	X =  251.204  mm,	Y =   -385.900  mm,	Z =   -311.265  mm,
	W =  90.000 deg,	P =   0.000 deg,	R =   90.000 deg
};
P[2440]{
   GP1:
	UF : 0, UT : 6,		CONFIG : 'N U T, 0, 0, 0',
	X =  250.053  mm,	Y =   -385.942  mm,	Z =   -320.068  mm,
	W =  90.000 deg,	P =   0.000 deg,	R =   90.000 deg
};
P[2441]{
   GP1:
	UF : 0, UT : 6,		CONFIG : 'N U T, 0, 0, 0',
	X =  249.566  mm,	Y =   -387.016  mm,	Z =   -309.000  mm,
	W =  90.000 deg,	P =   0.000 deg,	R =   90.000 deg
};
P[2442]{
   GP1:
	UF : 0, UT : 6,		CONFIG : 'N U T, 0, 0, 0',
	X =  248.771  mm,	Y =   -387.237  mm,	Z =   -309.100  mm,
	W =  90.000 deg,	P =   0.000 deg,	R =   90.000 deg
};
P[2443]{
   GP1:
	UF : 0, UT : 6,		CONFIG : 'N U T, 0, 0, 0',
	X =  247.127  mm,	Y =   -387.817  mm,	Z =   -310.009  mm,
	W =  90.000 deg,	P =   0.000 deg,	R =   90.000 deg
};
P[2444]{
   GP1:
	UF : 0, UT : 6,		CONFIG : 'N U T, 0, 0, 0',
	X =  246.328  mm,	Y =   -388.859  mm,	Z =   -309.000  mm,
	W =  90.000 deg,	P =   0.000 deg,	R =   90.000 deg
};
P[2445]{
   GP1:
	UF : 0, UT : 6,		CONFIG : 'N U T, 0, 0, 0',
	X =  245.729  mm,	Y =   -389.069  mm,	Z =   -324.841  mm,
	W =  90.000 deg,	P =   0.000 deg,	R =   90.000 deg
};
P[2446]{
   GP1:
	UF : 0, UT : 6,		CONFIG : 'N U T, 0, 0, 0',
	X =  244.982  mm,	Y =   -389.746  mm,	Z =   -309.100  mm,
	W =  90.000 deg,	P =   0.000 deg,	R =   90.000 deg
};
P[2447]{
   GP1:
	UF : 0, UT : 6,		CONFIG : 'N U T, 0, 0, 0',
	X =  243.856  mm,	Y =   -389.819  mm,	Z =   -309.100  mm,
	W =  90.000 deg,	P =   0.000 deg,	R =   90.000 deg
};
P[2448]{
   GP1:
	UF : 0, UT : 6,		CONFIG : 'N U T, 0, 0, 0',
	X =  243.235  mm,	Y =   -390.864  mm,	Z =   -309.100  mm,
	W =  90.000 deg,	P =   0.000 deg,	R =   90.000 deg
};
P[2449]{
   GP1:
	UF : 0, UT : 6,		CONFIG : 'N U T, 0, 0, 0',
	X =  242.193  mm,	Y =   -390.693  mm,	Z =   -309.000  mm,
	W =  90.000 deg,	P =   0.000 deg,	R =   90.000 deg
};
P[2450]{
   GP1:
	UF : 0, UT : 6,		CONFIG : 'N U T, 0, 0, 0',
	X =  241.203  mm,	Y =   -391.822  mm,	Z =   -309.100  mm,
	W =  90.000 deg,	P =   0.000 deg,	R =   90.000 deg
};
P[2451]{
   GP1:
	UF : 0, UT : 6,		CONFIG : 'N U T, 0, 0, 0',
	X =  240.398  mm,	Y =   -392.107  mm,	Z =   -309.000  mm,
	W =  90.000 deg,	P =   0.000 deg,	R =   90.000 deg
};
P[2452]{
   GP1:
	UF : 0, UT : 6,		CONFIG : 'N U T, 0, 0, 0',
	X =  239.660  mm,	Y =   -391.959  mm,	Z =   -309.100  mm,
	W =  90.000 deg,	P =   0.000 deg,	R =   90.000 deg
};
P[2453]{
   GP1:
	UF : 0, UT : 6,		CONFIG : 'N U T, 0, 0, 0',
	X =  238.993  mm,	Y =   -392.564  mm,	Z =   -309.000  mm,
	W =  90.000 deg,	P =   0.000 deg,	R =   90.000 deg
};
P[2454]{
   GP1:
	UF : 0, UT : 6,		CONFIG : 'N U T, 0, 0, 0',
	X =  238.146  mm,	Y =   -393.472  mm,	Z =   -309.000  mm,
	W =  90.000 deg,	P =   0.000 deg,	R =   90.000 deg
};
P[2455]{
   GP1:
	UF : 0, UT : 6,		CONFIG : 'N U T, 0, 0, 0',
	X =  236.954  mm,	Y =   -394.057  mm,	Z =   -309.000  mm,
	W =  90.000 deg,	P =   0.000 deg,	R =   90.000 deg
};
P[2456]{
   GP1:
	UF : 0, UT : 6,		CONFIG : 'N U T, 0, 0, 0',
	X =  236.048  mm,	Y =   -394.584  mm,	Z =   -309.100  mm,
	W =  90.000 deg,	P =   0.000 deg,	R =   90.000 deg
};
P[2457]{
   GP1:
	UF : 0, UT : 6,		CONFIG : 'N U T, 0, 0, 0',
	X =  235.652  mm,	Y =   -394.509  mm,	Z =   -309.100  mm,
	W =  90.000 deg,	P =   0.000 deg,	R =   90.000 deg
};
P[2458]{
   GP1:
	UF : 0, UT : 6,		CONFIG : 'N U T, 0, 0, 0',
	X =  235.672  mm,	Y =   -394.578  mm,	Z =   -309.000  mm,
	W =  90.000 deg,	P =   0.000 deg,	R =   90.000 deg
};
P[2459]{
   GP1:
	UF : 0, UT : 6,		CONFIG : 'N U T, 0, 0, 0',
	X =  235.717  mm,	Y =   -394.656  mm,	Z =   -309.100  mm,
	W =  90.000 deg,	P =   0.000 deg,	R =   90.000 deg
};
P[2460]{
   GP1:
	UF : 0, UT : 6,		CONFIG : 'N U T, 0, 0, 0',
	X =  235.797  mm,	Y =   -394.793  mm,	Z =   -309.100  mm,
	W =  90.000 deg,	P =   0.000 deg,	R =   90.000 deg
};
P[2461]{
   GP1:
	UF : 0, UT : 6,		CONFIG : 'N U T, 0, 0, 0',
	X =  235.811  mm,	Y =   -394.818  mm,	Z =   -309.000  mm,
	W =  90.000 deg,	P =   0.000 deg,	R =   90.000 deg
};
P[2462]{
   GP1:
	UF : 0, UT : 6,		CONFIG : 'N U T, 0, 0, 0',
	X =  235.830  mm,	Y =   -394.850  mm,	Z =   -309.000  mm,
	W =  90.000 deg,	P =   0.000 deg,	R =   90.000 deg
};
P[2463]{
   GP1:
	UF : 0, UT : 6,		CONFIG : 'N U T, 0, 0, 0',
	X =  235.853  mm,	Y =   -394.890  mm,	Z =   -309.000  mm,
	W =  90.000 deg,	P =   0.000 deg,	R =   90.000 deg
};
P[2464]{
   GP1:
	UF : 0, UT : 6,		CONFIG : 'N U T, 0, 0, 0',
	X =  235.853  mm,	Y =   -394.890  mm,	Z =   -309.100  mm,
	W =  90.000 deg,	P =   0.000 deg,	R =   90.000 deg
};
P[2465]{
   GP1:
	UF : 0, UT : 6,		CONFIG : 'N U T, 0, 0, 0',
	X =  235.932  mm,	Y =   -395.027  mm,	Z =   -309.000  mm,
	W =  90.000 deg,	P =   0.000 deg,	R =   90.000 deg
};
P[2466]{
   GP1:
	UF : 0, UT : 6,		CONFIG : 'N U T, 0, 0, 0',
	X =  234.712  mm,	Y =   -395.169  mm,	Z =   -311.663  mm,
	W =  90.000 deg,	P =   0.000 deg,	R =   90.000 deg
};
P[2467]{
   GP1:
	UF : 0, UT : 6,		CONFIG : 'N U T, 0, 0, 0',
	X =  233.900  mm,	Y =   -396.049  mm,	Z =   -309.000  mm,
	W =  90.000 deg,	P =   0.000 deg,	R =   90.000 deg
};
P[2468]{
   GP1:
	UF : 0, UT : 6,		CONFIG : 'N U T, 0, 0, 0',
	X =  232.847  mm,	Y =   -396.367  mm,	Z =   -309.000  mm,
	W =  90.000 deg,	P =   0.000 deg,	R =   90.000 deg
};
P[2469]{
   GP1:
	UF : 0, UT : 6,		CONFIG : 'N U T, 0, 0, 0',
	X =  231.860  mm,	Y =   -397.593  mm,	Z =   -322.086  mm,
	W =  90.000 deg,	P =   0.000 deg,	R =   90.000 deg
};
P[2470]{
   GP1:
	UF : 0, UT : 6,		CONFIG : 'N U T, 0, 0, 0',
	X =  231.255  mm,	Y =   -396.883  mm,	Z =   -309.100  mm,
	W =  90.000 deg,	P =   0.000 deg,	R =   90.000 deg
};
P[2471]{
   GP1:
	UF : 0, UT : 6,		CONFIG : 'N U T, 0, 0, 0',
	X =  230.508  mm,	Y =   -398.026  mm,	Z =   -309.100  mm,
	W =  90.000 deg,	P =   0.000 deg,	R =   90.000 deg
};
P[2472]{
   GP1:
	UF : 0, UT : 6,		CONFIG : 'N U T, 0, 0, 0',
	X =  229.295  mm,	Y =   -398.480  mm,	Z =   -309.000  mm,
	W =  90.000 deg,	P =   0.000 deg,	R =   90.000 deg
};
P[2473]{
   GP1:
	UF : 0, UT : 6,		CONFIG : 'N U T, 0, 0, 0',
	X =  228.271  mm,	Y =   -399.037  mm,	Z =   -309.100  mm,
	W =  90.000 deg,	P =   0.000 deg,	R =   90.000 deg
};
P[2474]{
   GP1:
	UF : 0, UT : 6,		CONFIG : 'N U T, 0, 0, 0',
	X =  227.431  mm,	Y =   -399.645  mm,	Z =   -309.000  mm,
	W =  90.000 deg,	P =   0.000 deg,	R =   90.000 deg
};
P[2475]{
   GP1:
	UF : 0, UT : 6,		CONFIG : 'N U T, 0, 0, 0',
	X =  227.107  mm,	Y =   -400.328  mm,	Z =   -309.000  mm,
	W =  90.000 deg,	P =   0.000 deg,	R =   90.000 deg
};
P[2476]{
   GP1:
	UF : 0, UT : 6,		CONFIG : 'N U T, 0, 0, 0',
	X =  226.158  mm,	Y =   -400.362  mm,	Z =   -309.000  mm,
	W =  90.000 deg,	P =   0.000 deg,	R =   90.000 deg
};
P[2477]{
   GP1:
	UF : 0, UT : 6,		CONFIG : 'N U T, 0, 0, 0',
	X =  225.458  mm,	Y =   -400.942  mm,	Z =   -309.100  mm,
	W =  90.000 deg,	P =   0.000 deg,	R =   90.000 deg
};
P[2478]{
   GP1:
	UF : 0, UT : 6,		CONFIG : 'N U T, 0, 0, 0',
	X =  223.961  mm,	Y =   -401.723  mm,	Z =   -309.000  mm,
	W =  90.000 deg,	P =   0.000 deg,	R =   90.000 deg
};
P[2479]{
   GP1:
	UF : 0, UT : 6,		CONFIG : 'N U T, 0, 0, 0',
	X =  222.266  mm,	Y =   -402.738  mm,	Z =   -309.000  mm,
	W =  90.000 deg,	P =   0.000 deg,	R =   90.000 deg
};
P[2480]{
   GP1:
	UF : 0, UT : 6,		CONFIG : 'N U T, 0, 0, 0',
	X =  221.544  mm,	Y =   -403.115  mm,	Z =   -309.000  mm,
	W =  90.000 deg,	P =   0.000 deg,	R =   90.000 deg
};
P[2481]{
   GP1:
	UF : 0, UT : 6,		CONFIG : 'N U T, 0, 0, 0',
	X =  220.694  mm,	Y =   -403.242  mm,	Z =   -309.100  mm,
	W =  90.000 deg,	P =   0.000 deg,	R =   90.000 deg
};
P[2482]{
   GP1:
	UF : 0, UT : 6,		CONFIG : 'N U T, 0, 0, 0',
	X =  220.123  mm,	Y =   -403.736  mm,	Z =   -309.000  mm,
	W =  90.000 deg,	P =   0.000 deg,	R =   90.000 deg
};
P[2483]{
   GP1:
	UF : 0, UT : 6,		CONFIG : 'N U T, 0, 0, 0',
	X =  218.860  mm,	Y =   -404.272  mm,	Z =   -309.000  mm,
	W =  90.000 deg,	P =   0.000 deg,	R =   90.000 deg
};
P[2484]{
   GP1:
	UF : 0, UT : 6,		CONFIG : 'N U T, 0, 0, 0',
	X =  217.826  mm,	Y =   -405.083  mm,	Z =   -309.000  mm,
	W =  90.000 deg,	P =   0.000 deg,	R =   90.000 deg
};
P[2485]{
   GP1:
	UF : 0, UT : 6,		CONFIG : 'N U T, 0, 0, 0',
	X =  217.425  mm,	Y =   -405.654  mm,	Z =   -309.100  mm,
	W =  90.000 deg,	P =   0.000 deg,	R =   90.000 deg
};
P[2486]{
   GP1:
	UF : 0, UT : 6,		CONFIG : 'N U T, 0, 0, 0',
	X =  216.186  mm,	Y =   -405.730  mm,	Z =   -309.000  mm,
	W =  90.000 deg,	P =   0.000 deg,	R =   90.000 deg
};
P[2487]{
   GP1:
	UF : 0, UT : 6,		CONFIG : 'N U T, 0, 0, 0',
	X =  215.322  mm,	Y =   -406.588  mm,	Z =   -309.000  mm,
	W =  90.000 deg,	P =   0.000 deg,	R =   90.000 deg
};
P[2488]{
   GP1:
	UF : 0, UT : 6,		CONFIG : 'N U T, 0, 0, 0',
	X =  214.425  mm,	Y =   -406.938  mm,	Z =   -309.000  mm,
	W =  90.000 deg,	P =   0.000 deg,	R =   90.000 deg
};
P[2489]{
   GP1:
	UF : 0, UT : 6,		CONFIG : 'N U T, 0, 0, 0',
	X =  212.907  mm,	Y =   -407.890  mm,	Z =   -309.000  mm,
	W =  90.000 deg,	P =   0.000 deg,	R =   90.000 deg
};
P[2490]{
   GP1:
	UF : 0, UT : 6,		CONFIG : 'N U T, 0, 0, 0',
	X =  212.273  mm,	Y =   -408.822  mm,	Z =   -309.000  mm,
	W =  90.000 deg,	P =   0.000 deg,	R =   90.000 deg
};
P[2491]{
   GP1:
	UF : 0, UT : 6,		CONFIG : 'N U T, 0, 0, 0',
	X =  211.523  mm,	Y =   -408.247  mm,	Z =   -309.840  mm,
	W =  90.000 deg,	P =   0.000 deg,	R =   90.000 deg
};
P[2492]{
   GP1:
	UF : 0, UT : 6,		CONFIG : 'N U T, 0, 0, 0',
	X =  211.810  mm,	Y =   -408.899  mm,	Z =   -309.000  mm,
	W =  90.000 deg,	P =   0.000 deg,	R =   90.000 deg
};
P[2493]{
   GP1:
	UF : 0, UT : 6,		CONFIG : 'N U T, 0, 0, 0',
	X =  211.264  mm,	Y =   -408.563  mm,	Z =   -309.000  mm,
	W =  90.000 deg,	P =   0.000 deg,	R =   90.000 deg
};
P[2494]{
   GP1:
	UF : 0, UT : 6,		CONFIG : 'N U T, 0, 0, 0',
	X =  211.213  mm,	Y =   -409.187  mm,	Z =   -309.100  mm,
	W =  90.000 deg,	P =   0.000 deg,	R =   90.000 deg
};
P[2495]{
   GP1:
	UF : 0, UT : 6,		CONFIG : 'N U T, 0, 0, 0',
	X =  210.542  mm,	Y =   -409.005  mm,	Z =   -309.000  mm,
	W =  90.000 deg,	P =   0.000 deg,	R =   90.000 deg
};
P[2496]{
   GP1:
	UF : 0, UT : 6,		CONFIG : 'N U T, 0, 0, 0',
	X =  210.183  mm,	Y =   -409.615  mm,	Z =   -311.087  mm,
	W =  90.000 deg,	P =   0.000 deg,	R =   90.000 deg
};
P[2497]{
   GP1:
	UF : 0, UT : 6,		CONFIG : 'N U T, 0, 0, 0',
	X =  209.312  mm,	Y =   -409.801  mm,	Z =   -309.000  mm,
	W =  90.000 deg,	P =   0.000 deg,	R =   90.000 deg
};
P[2498]{
   GP1:
	UF : 0, UT : 6,		CONFIG : 'N U T, 0, 0, 0',
	X =  208.830  mm,	Y =   -410.582  mm,	Z =   -326.834  mm,
	W =  90.000 deg,	P =   0.000 deg,	R =   90.000 deg
};
P[2499]{
   GP1:
	UF : 0, UT : 6,		CONFIG : 'N U T, 0, 0, 0',
	X =  207.578  mm,	Y =   -411.271  mm,	Z =   -319.896  mm,
	W =  90.000 deg,	P =   0.000 deg,	R =   90.000 deg
};
P[2500]{
   GP1:
	UF : 0, UT : 6,		CONFIG : 'N U T, 0, 0, 0',
	X =  206.272  mm,	Y =   -411.225  mm,	Z =   -309.000  mm,
	W =  90.000 deg,	P =   0.000 deg,	R =   90.000 deg
};
P[2501]{
   GP1:
	UF : 0, UT : 6,		CONFIG : 'N U T, 0, 0, 0',
	X =  205.768  mm,	Y =   -411.902  mm,	Z =   -309.000  mm,
	W =  90.000 deg,	P =   0.000 deg,	R =   90.000 deg
};
P[2502]{
   GP1:
	UF : 0, UT : 6,		CONFIG : 'N U T, 0, 0, 0',
	X =  205.135  mm,	Y =   -412.565  mm,	Z =   -309.000  mm,
	W =  90.000 deg,	P =   0.000 deg,	R =   90.000 deg
};
P[2503]{
   GP1:
	UF : 0, UT : 6,		CONFIG : 'N U T, 0, 0, 0',
	X =  204.079  mm,	Y =   -412.679  mm,	Z =   -309.000  mm,
	W =  90.000 deg,	P =   0.000 deg,	R =   90.000 deg
};
P[2504]{
   GP1:
	UF : 0, UT : 6,		CONFIG : 'N U T, 0, 0, 0',
	X =  203.955  mm,	Y =   -413.351  mm,	Z =   -309.000  mm,
	W =  90.000 deg,	P =   0.000 deg,	R =   90.000 deg
};
P[2505]{
   GP1:
	UF : 0, UT : 6,		CONFIG : 'N U T, 0, 0, 0',
	X =  203.212  mm,	Y =   -413.679  mm,	Z =   -309.100  mm,
	W =  90.000 deg,	P =   0.000 deg,	R =   90.000 deg
};
P[2506]{
   GP1:
	UF : 0, UT : 6,		CONFIG : 'N U T, 0, 0, 0',
	X =  201.743  mm,	Y =   -414.498  mm,	Z =   -320.312  mm,
	W =  90.000 deg,	P =   0.000 deg,	R =   90.000 deg
};
P[2507]{
   GP1:
	UF : 0, UT : 6,		CONFIG : 'N U T, 0, 0, 0',
	X =  200.955  mm,	Y =   -414.995  mm,	Z =   -309.100  mm,
	W =  90.000 deg,	P =   0.000 deg,	R =   90.000 deg
};
P[2508]{
   GP1:
	UF : 0, UT : 6,		CONFIG : 'N U T, 0, 0, 0',
	X =  199.958  mm,	Y =   -415.276  mm,	Z =   -309.000  mm,
	W =  90.000 deg,	P =   0.000 deg,	R =   90.000 deg
};
P[2509]{
   GP1:
	UF : 0, UT : 6,		CONFIG : 'N U T, 0, 0, 0',
	X =  199.292  mm,	Y =   -415.680  mm,	Z =   -309.000  mm,
	W =  90.000 deg,	P =   0.000 deg,	R =   90.000 deg
};
P[2510]{
   GP1:
	UF : 0, UT : 6,		CONFIG : 'N U T, 0, 0, 0',
	X =  198.614  mm,	Y =   -416.039  mm,	Z =   -309.000  mm,
	W =  90.000 deg,	P =   0.000 deg,	R =   90.000 deg
};
P[2511]{
   GP1:
	UF : 0, UT : 6,		CONFIG : 'N U T, 0, 0, 0',
	X =  197.853  mm,	Y =   -416.086  mm,	Z =   -309.100  mm,
	W =  90.000 deg,	P =   0.000 deg,	R =   90.000 deg
};
P[2512]{
   GP1:
	UF : 0, UT : 6,		CONFIG : 'N U T, 0, 0, 0',
	X =  197.431  mm,	Y =   -416.630  mm,	Z =   -309.000  mm,
	W =  90.000 deg,	P =   0.000 deg,	R =   90.000 deg
};
P[2513]{
   GP1:
	UF : 0, UT : 6,		CONFIG : 'N U T, 0, 0, 0',
	X =  197.048  mm,	Y =   -417.376  mm,	Z =   -309.000  mm,
	W =  90.000 deg,	P =   0.000 deg,	R =   90.000 deg
};
P[2514]{
   GP1:
	UF : 0, UT : 6,		CONFIG : 'N U T, 0, 0, 0',
	X =  195.899  mm,	Y =   -417.317  mm,	Z =   -309.100  mm,
	W =  90.000 deg,	P =   0.000 deg,	R =   90.000 deg
};
P[2515]{
   GP1:
	UF : 0, UT : 6,		CONFIG : 'N U T, 0, 0, 0',
	X =  195.162  mm,	Y =   -418.086  mm,	Z =   -309.769  mm,
	W =  90.000 deg,	P =   0.000 deg,	R =   90.000 deg
};
P[2516]{
   GP1:
	UF : 0, UT : 6,		CONFIG : 'N U T, 0, 0, 0',
	X =  193.868  mm,	Y =   -419.148  mm,	Z =   -320.299  mm,
	W =  90.000 deg,	P =   0.000 deg,	R =   90.000 deg
};
P[2517]{
   GP1:
	UF : 0, UT : 6,		CONFIG : 'N U T, 0, 0, 0',
	X =  192.981  mm,	Y =   -419.724  mm,	Z =   -309.000  mm,
	W =  90.000 deg,	P =   0.000 deg,	R =   90.000 deg
};
P[2518]{
   GP1:
	UF : 0, UT : 6,		CONFIG : 'N U T, 0, 0, 0',
	X =  191.775  mm,	Y =   -420.224  mm,	Z =   -309.100  mm,
	W =  90.000 deg,	P =   0.000 deg,	R =   90.000 deg
};
P[2519]{
   GP1:
	UF : 0, UT : 6,		CONFIG : 'N U T, 0, 0, 0',
	X =  190.726  mm,	Y =   -420.304  mm,	Z =   -309.000  mm,
	W =  90.000 deg,	P =   0.000 deg,	R =   90.000 deg
};
P[2520]{
   GP1:
	UF : 0, UT : 6,		CONFIG : 'N U T, 0, 0, 0',
	X =  191.173  mm,	Y =   -421.086  mm,	Z =   -309.000  mm,
	W =  90.000 deg,	P =   0.000 deg,	R =   90.000 deg
};
P[2521]{
   GP1:
	UF : 0, UT : 6,		CONFIG : 'N U T, 0, 0, 0',
	X =  190.334  mm,	Y =   -421.290  mm,	Z =   -322.014  mm,
	W =  90.000 deg,	P =   0.000 deg,	R =   90.000 deg
};
P[2522]{
   GP1:
	UF : 0, UT : 6,		CONFIG : 'N U T, 0, 0, 0',
	X =  189.270  mm,	Y =   -421.536  mm,	Z =   -309.000  mm,
	W =  90.000 deg,	P =   0.000 deg,	R =   90.000 deg
};
P[2523]{
   GP1:
	UF : 0, UT : 6,		CONFIG : 'N U T, 0, 0, 0',
	X =  187.988  mm,	Y =   -422.472  mm,	Z =   -309.000  mm,
	W =  90.000 deg,	P =   0.000 deg,	R =   90.000 deg
};
P[2524]{
   GP1:
	UF : 0, UT : 6,		CONFIG : 'N U T, 0, 0, 0',
	X =  186.884  mm,	Y =   -422.846  mm,	Z =   -309.000  mm,
	W =  90.000 deg,	P =   0.000 deg,	R =   90.000 deg
};
P[2525]{
   GP1:
	UF : 0, UT : 6,		CONFIG : 'N U T, 0, 0, 0',
	X =  186.127  mm,	Y =   -423.764  mm,	Z =   -309.000  mm,
	W =  90.000 deg,	P =   0.000 deg,	R =   90.000 deg
};
P[2526]{
   GP1:
	UF : 0, UT : 6,		CONFIG : 'N U T, 0, 0, 0',
	X =  184.971  mm,	Y =   -424.213  mm,	Z =   -309.000  mm,
	W =  90.000 deg,	P =   0.000 deg,	R =   90.000 deg
};
P[2527]{
   GP1:
	UF : 0, UT : 6,		CONFIG : 'N U T, 0, 0, 0',
	X =  184.314  mm,	Y =   -424.591  mm,	Z =   -309.000  mm,
	W =  90.000 deg,	P =   0.000 deg,	R =   90.000 deg
};
P[2528]{
   GP1:
	UF : 0, UT : 6,		CONFIG : 'N U T, 0, 0, 0',
	X =  182.781  mm,	Y =   -425.363  mm,	Z =   -309.000  mm,
	W =  90.000 deg,	P =   0.000 deg,	R =   90.000 deg
};
P[2529]{
   GP1:
	UF : 0, UT : 6,		CONFIG : 'N U T, 0, 0, 0',
	X =  181.660  mm,	Y =   -425.576  mm,	Z =   -309.100  mm,
	W =  90.000 deg,	P =   0.000 deg,	R =   90.000 deg
};
P[2530]{
   GP1:
	UF : 0, UT : 6,		CONFIG : 'N U T, 0, 0, 0',
	X =  181.249  mm,	Y =   -426.623  mm,	Z =   -309.000  mm,
	W =  90.000 deg,	P =   0.000 deg,	R =   90.000 deg
};
P[2531]{
   GP1:
	UF : 0, UT : 6,		CONFIG : 'N U T, 0, 0, 0',
	X =  180.447  mm,	Y =   -426.800  mm,	Z =   -309.000  mm,
	W =  90.000 deg,	P =   0.000 deg,	R =   90.000 deg
};
P[2532]{
   GP1:
	UF : 0, UT : 6,		CONFIG : 'N U T, 0, 0, 0',
	X =  179.771  mm,	Y =   -426.566  mm,	Z =   -309.000  mm,
	W =  90.000 deg,	P =   0.000 deg,	R =   90.000 deg
};
P[2533]{
   GP1:
	UF : 0, UT : 6,		CONFIG : 'N U T, 0, 0, 0',
	X =  179.286  mm,	Y =   -427.366  mm,	Z =   -309.000  mm,
	W =  90.000 deg,	P =   0.000 deg,	R =   90.000 deg
};
P[2534]{
   GP1:
	UF : 0, UT : 6,		CONFIG : 'N U T, 0, 0, 0',
	X =  178.106  mm,	Y =   -427.866  mm,	Z =   -309.100  mm,
	W =  90.000 deg,	P =   0.000 deg,	R =   90.000 deg
};
P[2535]{
   GP1:
	UF : 0, UT : 6,		CONFIG : 'N U T, 0, 0, 0',
	X =  177.596  mm,	Y =   -428.277  mm,	Z =   -309.000  mm,
	W =  90.000 deg,	P =   0.000 deg,	R =   90.000 deg
};
P[2536]{
   GP1:
	UF : 0, UT : 6,		CONFIG : 'N U T, 0, 0, 0',
	X =  176.414  mm,	Y =   -428.917  mm,	Z =   -309.000  mm,
	W =  90.000 deg,	P =   0.000 deg,	R =   90.000 deg
};
P[2537]{
   GP1:
	UF : 0, UT : 6,		CONFIG : 'N U T, 0, 0, 0',
	X =  175.410  mm,	Y =   -429.586  mm,	Z =   -309.000  mm,
	W =  90.000 deg,	P =   0.000 deg,	R =   90.000 deg
};
P[2538]{
   GP1:
	UF : 0, UT : 6,		CONFIG : 'N U T, 0, 0, 0',
	X =  174.790  mm,	Y =   -430.203  mm,	Z =   -309.100  mm,
	W =  90.000 deg,	P =   0.000 deg,	R =   90.000 deg
};
P[2539]{
   GP1:
	UF : 0, UT : 6,		CONFIG : 'N U T, 0, 0, 0',
	X =  174.023  mm,	Y =   -430.329  mm,	Z =   -309.000  mm,
	W =  90.000 deg,	P =   0.000 deg,	R =   90.000 deg
};
P[2540]{
   GP1:
	UF : 0, UT : 6,		CONFIG : 'N U T, 0, 0, 0',
	X =  173.246  mm,	Y =   -430.866  mm,	Z =   -309.000  mm,
	W =  90.000 deg,	P =   0.000 deg,	R =   90.000 deg
};
P[2541]{
   GP1:
	UF : 0, UT : 6,		CONFIG : 'N U T, 0, 0, 0',
	X =  172.207  mm,	Y =   -431.345  mm,	Z =   -309.000  mm,
	W =  90.000 deg,	P =   0.000 deg,	R =   90.000 deg
};
P[2542]{
   GP1:
	UF : 0, UT : 6,		CONFIG : 'N U T, 0, 0, 0',
	X =  171.867  mm,	Y =   -432.022  mm,	Z =   -309.000  mm,
	W =  90.000 deg,	P =   0.000 deg,	R =   90.000 deg
};
P[2543]{
   GP1:
	UF : 0, UT : 6,		CONFIG : 'N U T, 0, 0, 0',
	X =  170.157  mm,	Y =   -432.977  mm,	Z =   -309.000  mm,
	W =  90.000 deg,	P =   0.000 deg,	R =   90.000 deg
};
P[2544]{
   GP1:
	UF : 0, UT : 6,		CONFIG : 'N U T, 0, 0, 0',
	X =  169.135  mm,	Y =   -432.828  mm,	Z =   -309.000  mm,
	W =  90.000 deg,	P =   0.000 deg,	R =   90.000 deg
};
P[2545]{
   GP1:
	UF : 0, UT : 6,		CONFIG : 'N U T, 0, 0, 0',
	X =  168.495  mm,	Y =   -433.303  mm,	Z =   -309.000  mm,
	W =  90.000 deg,	P =   0.000 deg,	R =   90.000 deg
};
P[2546]{
   GP1:
	UF : 0, UT : 6,		CONFIG : 'N U T, 0, 0, 0',
	X =  168.424  mm,	Y =   -434.070  mm,	Z =   -309.000  mm,
	W =  90.000 deg,	P =   0.000 deg,	R =   90.000 deg
};
P[2547]{
   GP1:
	UF : 0, UT : 6,		CONFIG : 'N U T, 0, 0, 0',
	X =  166.498  mm,	Y =   -434.623  mm,	Z =   -309.000  mm,
	W =  90.000 deg,	P =   0.000 deg,	R =   90.000 deg
};
P[2548]{
   GP1:
	UF : 0, UT : 6,		CONFIG : 'N U T, 0, 0, 0',
	X =  165.399  mm,	Y =   -435.440  mm,	Z =   -309.000  mm,
	W =  90.000 deg,	P =   0.000 deg,	R =   90.000 deg
};
P[2549]{
   GP1:
	UF : 0, UT : 6,		CONFIG : 'N U T, 0, 0, 0',
	X =  164.602  mm,	Y =   -435.687  mm,	Z =   -309.000  mm,
	W =  90.000 deg,	P =   0.000 deg,	R =   90.000 deg
};
P[2550]{
   GP1:
	UF : 0, UT : 6,		CONFIG : 'N U T, 0, 0, 0',
	X =  163.906  mm,	Y =   -436.668  mm,	Z =   -309.000  mm,
	W =  90.000 deg,	P =   0.000 deg,	R =   90.000 deg
};
P[2551]{
   GP1:
	UF : 0, UT : 6,		CONFIG : 'N U T, 0, 0, 0',
	X =  162.841  mm,	Y =   -437.088  mm,	Z =   -309.100  mm,
	W =  90.000 deg,	P =   0.000 deg,	R =   90.000 deg
};
P[2552]{
   GP1:
	UF : 0, UT : 6,		CONFIG : 'N U T, 0, 0, 0',
	X =  161.989  mm,	Y =   -437.881  mm,	Z =   -309.893  mm,
	W =  90.000 deg,	P =   0.000 deg,	R =   90.000 deg
};
P[2553]{
   GP1:
	UF : 0, UT : 6,		CONFIG : 'N U T, 0, 0, 0',
	X =  161.304  mm,	Y =   -437.408  mm,	Z =   -309.000  mm,
	W =  90.000 deg,	P =   0.000 deg,	R =   90.000 deg
};
P[2554]{
   GP1:
	UF : 0, UT : 6,		CONFIG : 'N U T, 0, 0, 0',
	X =  160.368  mm,	Y =   -438.644  mm,	Z =   -309.000  mm,
	W =  90.000 deg,	P =   0.000 deg,	R =   90.000 deg
};
P[2555]{
   GP1:
	UF : 0, UT : 6,		CONFIG : 'N U T, 0, 0, 0',
	X =  159.528  mm,	Y =   -438.648  mm,	Z =   -309.000  mm,
	W =  90.000 deg,	P =   0.000 deg,	R =   90.000 deg
};
P[2556]{
   GP1:
	UF : 0, UT : 6,		CONFIG : 'N U T, 0, 0, 0',
	X =  158.573  mm,	Y =   -439.371  mm,	Z =   -309.000  mm,
	W =  90.000 deg,	P =   0.000 deg,	R =   90.000 deg
};
P[2557]{
   GP1:
	UF : 0, UT : 6,		CONFIG : 'N U T, 0, 0, 0',
	X =  157.879  mm,	Y =   -440.242  mm,	Z =   -309.000  mm,
	W =  90.000 deg,	P =   0.000 deg,	R =   90.000 deg
};
P[2558]{
   GP1:
	UF : 0, UT : 6,		CONFIG : 'N U T, 0, 0, 0',
	X =  157.140  mm,	Y =   -440.386  mm,	Z =   -309.000  mm,
	W =  90.000 deg,	P =   0.000 deg,	R =   90.000 deg
};
P[2559]{
   GP1:
	UF : 0, UT : 6,		CONFIG : 'N U T, 0, 0, 0',
	X =  156.396  mm,	Y =   -440.305  mm,	Z =   -309.000  mm,
	W =  90.000 deg,	P =   0.000 deg,	R =   90.000 deg
};
P[2560]{
   GP1:
	UF : 0, UT : 6,		CONFIG : 'N U T, 0, 0, 0',
	X =  155.713  mm,	Y =   -441.118  mm,	Z =   -309.000  mm,
	W =  90.000 deg,	P =   0.000 deg,	R =   90.000 deg
};
P[2561]{
   GP1:
	UF : 0, UT : 6,		CONFIG : 'N U T, 0, 0, 0',
	X =  155.008  mm,	Y =   -441.324  mm,	Z =   -309.000  mm,
	W =  90.000 deg,	P =   0.000 deg,	R =   90.000 deg
};
P[2562]{
   GP1:
	UF : 0, UT : 6,		CONFIG : 'N U T, 0, 0, 0',
	X =  154.353  mm,	Y =   -441.739  mm,	Z =   -309.000  mm,
	W =  90.000 deg,	P =   0.000 deg,	R =   90.000 deg
};
P[2563]{
   GP1:
	UF : 0, UT : 6,		CONFIG : 'N U T, 0, 0, 0',
	X =  153.918  mm,	Y =   -442.344  mm,	Z =   -309.000  mm,
	W =  90.000 deg,	P =   0.000 deg,	R =   90.000 deg
};
P[2564]{
   GP1:
	UF : 0, UT : 6,		CONFIG : 'N U T, 0, 0, 0',
	X =  153.557  mm,	Y =   -442.273  mm,	Z =   -309.000  mm,
	W =  90.000 deg,	P =   0.000 deg,	R =   90.000 deg
};
P[2565]{
   GP1:
	UF : 0, UT : 6,		CONFIG : 'N U T, 0, 0, 0',
	X =  153.337  mm,	Y =   -441.968  mm,	Z =   -309.000  mm,
	W =  90.000 deg,	P =   0.000 deg,	R =   90.000 deg
};
P[2566]{
   GP1:
	UF : 0, UT : 6,		CONFIG : 'N U T, 0, 0, 0',
	X =  153.390  mm,	Y =   -442.061  mm,	Z =   -309.100  mm,
	W =  90.000 deg,	P =   0.000 deg,	R =   90.000 deg
};
P[2567]{
   GP1:
	UF : 0, UT : 6,		CONFIG : 'N U T, 0, 0, 0',
	X =  153.417  mm,	Y =   -442.107  mm,	Z =   -309.100  mm,
	W =  90.000 deg,	P =   0.000 deg,	R =   90.000 deg
};
P[2568]{
   GP1:
	UF : 0, UT : 6,		CONFIG : 'N U T, 0, 0, 0',
	X =  153.429  mm,	Y =   -442.129  mm,	Z =   -309.000  mm,
	W =  90.000 deg,	P =   0.000 deg,	R =   90.000 deg
};
P[2569]{
   GP1:
	UF : 0, UT : 6,		CONFIG : 'N U T, 0, 0, 0',
	X =  153.499  mm,	Y =   -442.250  mm,	Z =   -309.000  mm,
	W =  90.000 deg,	P =   0.000 deg,	R =   90.000 deg
};
P[2570]{
   GP1:
	UF : 0, UT : 6,		CONFIG : 'N U T, 0, 0, 0',
	X =  153.512  mm,	Y =   -442.271  mm,	Z =   -309.000  mm,
	W =  90.000 deg,	P =   0.000 deg,	R =   90.000 deg
};
P[2571]{
   GP1:
	UF : 0, UT : 6,		CONFIG : 'N U T, 0, 0, 0',
	X =  153.675  mm,	Y =   -442.554  mm,	Z =   -309.000  mm,
	W =  90.000 deg,	P =   0.000 deg,	R =   90.000 deg
};
P[2572]{
   GP1:
	UF : 0, UT : 6,		CONFIG : 'N U T, 0, 0, 0',
	X =  153.676  mm,	Y =   -442.556  mm,	Z =   -309.100  mm,
	W =  90.000 deg,	P =   0.000 deg,	R =   90.000 deg
};
P[2573]{
   GP1:
	UF : 0, UT : 6,		CONFIG : 'N U T, 0, 0, 0',
	X =  153.700  mm,	Y =   -442.598  mm,	Z =   -309.000  mm,
	W =  90.000 deg,	P =   0.000 deg,	R =   90.000 deg
};
P[2574]{
   GP1:
	UF : 0, UT : 6,		CONFIG : 'N U T, 0, 0, 0',
	X =  153.197  mm,	Y =   -442.479  mm,	Z =   -309.100  mm,
	W =  90.000 deg,	P =   0.000 deg,	R =   90.000 deg
};
P[2575]{
   GP1:
	UF : 0, UT : 6,		CONFIG : 'N U T, 0, 0, 0',
	X =  151.809  mm,	Y =   -442.696  mm,	Z =   -309.000  mm,
	W =  90.000 deg,	P =   0.000 deg,	R =   90.000 deg
};
P[2576]{
   GP1:
	UF : 0, UT : 6,		CONFIG : 'N U T, 0, 0, 0',
	X =  151.136  mm,	Y =   -443.692  mm,	Z =   -319.431  mm,
	W =  90.000 deg,	P =   0.000 deg,	R =   90.000 deg
};
P[2577]{
   GP1:
	UF : 0, UT : 6,		CONFIG : 'N U T, 0, 0, 0',
	X =  150.368  mm,	Y =   -444.081  mm,	Z =   -309.000  mm,
	W =  90.000 deg,	P =   0.000 deg,	R =   90.000 deg
};
P[2578]{
   GP1:
	UF : 0, UT : 6,		CONFIG : 'N U T, 0, 0, 0',
	X =  149.653  mm,	Y =   -444.476  mm,	Z =   -309.000  mm,
	W =  90.000 deg,	P =   0.000 deg,	R =   90.000 deg
};
P[2579]{
   GP1:
	UF : 0, UT : 6,		CONFIG : 'N U T, 0, 0, 0',
	X =  148.623  mm,	Y =   -444.808  mm,	Z =   -309.000  mm,
	W =  90.000 deg,	P =   0.000 deg,	R =   90.000 deg
};
P[2580]{
   GP1:
	UF : 0, UT : 6,		CONFIG : 'N U T, 0, 0, 0',
	X =  147.296  mm,	Y =   -446.099  mm,	Z =   -309.000  mm,
	W =  90.000 deg,	P =   0.000 deg,	R =   90.000 deg
};
P[2581]{
   GP1:
	UF : 0, UT : 6,		CONFIG : 'N U T, 0, 0, 0',
	X =  146.188  mm,	Y =   -446.215  mm,	Z =   -309.000  mm,
	W =  90.000 deg,	P =   0.000 deg,	R =   90.000 deg
};
P[2582]{
   GP1:
	UF : 0, UT : 6,		CONFIG : 'N U T, 0, 0, 0',
	X =  145.216  mm,	Y =   -446.906  mm,	Z =   -309.100  mm,
	W =  90.000 deg,	P =   0.000 deg,	R =   90.000 deg
};
P[2583]{
   GP1:
	UF : 0, UT : 6,		CONFIG : 'N U T, 0, 0, 0',
	X =  144.453  mm,	Y =   -447.564  mm,	Z =   -309.000  mm,
	W =  90.000 deg,	P =   0.000 deg,	R =   90.000 deg
};
P[2584]{
   GP1:
	UF : 0, UT : 6,		CONFIG : 'N U T, 0, 0, 0',
	X =  143.642  mm,	Y =   -447.566  mm,	Z =   -309.100  mm,
	W =  90.000 deg,	P =   0.000 deg,	R =   90.000 deg
};
P[2585]{
   GP1:
	UF : 0, UT : 6,		CONFIG : 'N U T, 0, 0, 0',
	X =  142.855  mm,	Y =   -448.215  mm,	Z =   -309.000  mm,
	W =  90.000 deg,	P =   0.000 deg,	R =   90.000 deg
};
P[2586]{
   GP1:
	UF : 0, UT : 6,		CONFIG : 'N U T, 0, 0, 0',
	X =  141.854  mm,	Y =   -449.026  mm,	Z =   -309.000  mm,
	W =  90.000 deg,	P =   0.000 deg,	R =   90.000 deg
};
P[2587]{
   GP1:
	UF : 0, UT : 6,		CONFIG : 'N U T, 0, 0, 0',
	X =  140.839  mm,	Y =   -449.789  mm,	Z =   -309.000  mm,
	W =  90.000 deg,	P =   0.000 deg,	R =   90.000 deg
};
P[2588]{
   GP1:
	UF : 0, UT : 6,		CONFIG : 'N U T, 0, 0, 0',
	X =  139.971  mm,	Y =   -449.754  mm,	Z =   -316.099  mm,
	W =  90.000 deg,	P =   0.000 deg,	R =   90.000 deg
};
P[2589]{
   GP1:
	UF : 0, UT : 6,		CONFIG : 'N U T, 0, 0, 0',
	X =  139.488  mm,	Y =   -450.789  mm,	Z =   -309.100  mm,
	W =  90.000 deg,	P =   0.000 deg,	R =   90.000 deg
};
P[2590]{
   GP1:
	UF : 0, UT : 6,		CONFIG : 'N U T, 0, 0, 0',
	X =  138.483  mm,	Y =   -450.497  mm,	Z =   -309.000  mm,
	W =  90.000 deg,	P =   0.000 deg,	R =   90.000 deg
};
P[2591]{
   GP1:
	UF : 0, UT : 6,		CONFIG : 'N U T, 0, 0, 0',
	X =  145.995  mm,	Y =   -463.381  mm,	Z =   -309.000  mm,
	W =  90.000 deg,	P =   0.000 deg,	R =   90.000 deg
};
P[2592]{
   GP1:
	UF : 0, UT : 6,		CONFIG : 'N U T, 0, 0, 0',
	X =  146.551  mm,	Y =   -464.097  mm,	Z =   -309.100  mm,
	W =  90.000 deg,	P =   0.000 deg,	R =   90.000 deg
};
P[2593]{
   GP1:
	UF : 0, UT : 6,		CONFIG : 'N U T, 0, 0, 0',
	X =  147.925  mm,	Y =   -463.215  mm,	Z =   -309.000  mm,
	W =  90.000 deg,	P =   0.000 deg,	R =   90.000 deg
};
P[2594]{
   GP1:
	UF : 0, UT : 6,		CONFIG : 'N U T, 0, 0, 0',
	X =  148.470  mm,	Y =   -462.667  mm,	Z =   -309.100  mm,
	W =  90.000 deg,	P =   0.000 deg,	R =   90.000 deg
};
P[2595]{
   GP1:
	UF : 0, UT : 6,		CONFIG : 'N U T, 0, 0, 0',
	X =  149.101  mm,	Y =   -461.749  mm,	Z =   -309.000  mm,
	W =  90.000 deg,	P =   0.000 deg,	R =   90.000 deg
};
P[2596]{
   GP1:
	UF : 0, UT : 6,		CONFIG : 'N U T, 0, 0, 0',
	X =  150.290  mm,	Y =   -461.267  mm,	Z =   -309.000  mm,
	W =  90.000 deg,	P =   0.000 deg,	R =   90.000 deg
};
P[2597]{
   GP1:
	UF : 0, UT : 6,		CONFIG : 'N U T, 0, 0, 0',
	X =  151.468  mm,	Y =   -461.033  mm,	Z =   -309.000  mm,
	W =  90.000 deg,	P =   0.000 deg,	R =   90.000 deg
};
P[2598]{
   GP1:
	UF : 0, UT : 6,		CONFIG : 'N U T, 0, 0, 0',
	X =  151.905  mm,	Y =   -460.393  mm,	Z =   -309.000  mm,
	W =  90.000 deg,	P =   0.000 deg,	R =   90.000 deg
};
P[2599]{
   GP1:
	UF : 0, UT : 6,		CONFIG : 'N U T, 0, 0, 0',
	X =  153.004  mm,	Y =   -459.500  mm,	Z =   -309.000  mm,
	W =  90.000 deg,	P =   0.000 deg,	R =   90.000 deg
};
P[2600]{
   GP1:
	UF : 0, UT : 6,		CONFIG : 'N U T, 0, 0, 0',
	X =  153.819  mm,	Y =   -459.457  mm,	Z =   -309.000  mm,
	W =  90.000 deg,	P =   0.000 deg,	R =   90.000 deg
};
P[2601]{
   GP1:
	UF : 0, UT : 6,		CONFIG : 'N U T, 0, 0, 0',
	X =  154.610  mm,	Y =   -459.138  mm,	Z =   -309.000  mm,
	W =  90.000 deg,	P =   0.000 deg,	R =   90.000 deg
};
P[2602]{
   GP1:
	UF : 0, UT : 6,		CONFIG : 'N U T, 0, 0, 0',
	X =  155.268  mm,	Y =   -458.821  mm,	Z =   -309.000  mm,
	W =  90.000 deg,	P =   0.000 deg,	R =   90.000 deg
};
P[2603]{
   GP1:
	UF : 0, UT : 6,		CONFIG : 'N U T, 0, 0, 0',
	X =  156.649  mm,	Y =   -458.328  mm,	Z =   -309.000  mm,
	W =  90.000 deg,	P =   0.000 deg,	R =   90.000 deg
};
P[2604]{
   GP1:
	UF : 0, UT : 6,		CONFIG : 'N U T, 0, 0, 0',
	X =  157.093  mm,	Y =   -457.489  mm,	Z =   -309.000  mm,
	W =  90.000 deg,	P =   0.000 deg,	R =   90.000 deg
};
P[2605]{
   GP1:
	UF : 0, UT : 6,		CONFIG : 'N U T, 0, 0, 0',
	X =  158.076  mm,	Y =   -457.124  mm,	Z =   -309.100  mm,
	W =  90.000 deg,	P =   0.000 deg,	R =   90.000 deg
};
P[2606]{
   GP1:
	UF : 0, UT : 6,		CONFIG : 'N U T, 0, 0, 0',
	X =  159.188  mm,	Y =   -456.288  mm,	Z =   -309.000  mm,
	W =  90.000 deg,	P =   0.000 deg,	R =   90.000 deg
};
P[2607]{
   GP1:
	UF : 0, UT : 6,		CONFIG : 'N U T, 0, 0, 0',
	X =  160.131  mm,	Y =   -455.836  mm,	Z =   -326.220  mm,
	W =  90.000 deg,	P =   0.000 deg,	R =   90.000 deg
};
P[2608]{
   GP1:
	UF : 0, UT : 6,		CONFIG : 'N U T, 0, 0, 0',
	X =  160.645  mm,	Y =   -455.321  mm,	Z =   -309.000  mm,
	W =  90.000 deg,	P =   0.000 deg,	R =   90.000 deg
};
P[2609]{
   GP1:
	UF : 0, UT : 6,		CONFIG : 'N U T, 0, 0, 0',
	X =  160.776  mm,	Y =   -454.852  mm,	Z =   -309.000  mm,
	W =  90.000 deg,	P =   0.000 deg,	R =   90.000 deg
};
P[2610]{
   GP1:
	UF : 0, UT : 6,		CONFIG : 'N U T, 0, 0, 0',
	X =  160.874  mm,	Y =   -455.023  mm,	Z =   -309.000  mm,
	W =  90.000 deg,	P =   0.000 deg,	R =   90.000 deg
};
P[2611]{
   GP1:
	UF : 0, UT : 6,		CONFIG : 'N U T, 0, 0, 0',
	X =  161.012  mm,	Y =   -455.261  mm,	Z =   -309.000  mm,
	W =  90.000 deg,	P =   0.000 deg,	R =   90.000 deg
};
P[2612]{
   GP1:
	UF : 0, UT : 6,		CONFIG : 'N U T, 0, 0, 0',
	X =  161.170  mm,	Y =   -455.535  mm,	Z =   -323.817  mm,
	W =  90.000 deg,	P =   0.000 deg,	R =   90.000 deg
};
P[2613]{
   GP1:
	UF : 0, UT : 6,		CONFIG : 'N U T, 0, 0, 0',
	X =  161.196  mm,	Y =   -455.579  mm,	Z =   -309.000  mm,
	W =  90.000 deg,	P =   0.000 deg,	R =   90.000 deg
};
P[2614]{
   GP1:
	UF : 0, UT : 6,		CONFIG : 'N U T, 0, 0, 0',
	X =  161.319  mm,	Y =   -455.634  mm,	Z =   -309.000  mm,
	W =  90.000 deg,	P =   0.000 deg,	R =   90.000 deg
};
P[2615]{
   GP1:
	UF : 0, UT : 6,		CONFIG : 'N U T, 0, 0, 0',
	X =  161.348  mm,	Y =   -455.458  mm,	Z =   -320.213  mm,
	W =  90.000 deg,	P =   0.000 deg,	R =   90.000 deg
};
P[2616]{
   GP1:
	UF : 0, UT : 6,		CONFIG : 'N U T, 0, 0, 0',
	X =  161.544  mm,	Y =   -455.141  mm,	Z =   -309.000  mm,
	W =  90.000 deg,	P =   0.000 deg,	R =   90.000 deg
};
P[2617]{
   GP1:
	UF : 0, UT : 6,		CONFIG : 'N U T, 0, 0, 0',
	X =  162.378  mm,	Y =   -455.021  mm,	Z =   -309.000  mm,
	W =  90.000 deg,	P =   0.000 deg,	R =   90.000 deg
};
P[2618]{
   GP1:
	UF : 0, UT : 6,		CONFIG : 'N U T, 0, 0, 0',
	X =  162.287  mm,	Y =   -454.506  mm,	Z =   -309.000  mm,
	W =  90.000 deg,	P =   0.000 deg,	R =   90.000 deg
};
P[2619]{
   GP1:
	UF : 0, UT : 6,		CONFIG : 'N U T, 0, 0, 0',
	X =  163.627  mm,	Y =   -453.962  mm,	Z =   -309.100  mm,
	W =  90.000 deg,	P =   0.000 deg,	R =   90.000 deg
};
P[2620]{
   GP1:
	UF : 0, UT : 6,		CONFIG : 'N U T, 0, 0, 0',
	X =  163.935  mm,	Y =   -453.268  mm,	Z =   -309.000  mm,
	W =  90.000 deg,	P =   0.000 deg,	R =   90.000 deg
};
P[2621]{
   GP1:
	UF : 0, UT : 6,		CONFIG : 'N U T, 0, 0, 0',
	X =  165.103  mm,	Y =   -453.333  mm,	Z =   -309.000  mm,
	W =  90.000 deg,	P =   0.000 deg,	R =   90.000 deg
};
P[2622]{
   GP1:
	UF : 0, UT : 6,		CONFIG : 'N U T, 0, 0, 0',
	X =  165.859  mm,	Y =   -452.501  mm,	Z =   -309.000  mm,
	W =  90.000 deg,	P =   0.000 deg,	R =   90.000 deg
};
P[2623]{
   GP1:
	UF : 0, UT : 6,		CONFIG : 'N U T, 0, 0, 0',
	X =  166.358  mm,	Y =   -451.819  mm,	Z =   -309.000  mm,
	W =  90.000 deg,	P =   0.000 deg,	R =   90.000 deg
};
P[2624]{
   GP1:
	UF : 0, UT : 6,		CONFIG : 'N U T, 0, 0, 0',
	X =  166.887  mm,	Y =   -452.114  mm,	Z =   -309.100  mm,
	W =  90.000 deg,	P =   0.000 deg,	R =   90.000 deg
};
P[2625]{
   GP1:
	UF : 0, UT : 6,		CONFIG : 'N U T, 0, 0, 0',
	X =  167.686  mm,	Y =   -451.512  mm,	Z =   -309.000  mm,
	W =  90.000 deg,	P =   0.000 deg,	R =   90.000 deg
};
P[2626]{
   GP1:
	UF : 0, UT : 6,		CONFIG : 'N U T, 0, 0, 0',
	X =  168.463  mm,	Y =   -450.699  mm,	Z =   -309.000  mm,
	W =  90.000 deg,	P =   0.000 deg,	R =   90.000 deg
};
P[2627]{
   GP1:
	UF : 0, UT : 6,		CONFIG : 'N U T, 0, 0, 0',
	X =  169.291  mm,	Y =   -450.860  mm,	Z =   -309.000  mm,
	W =  90.000 deg,	P =   0.000 deg,	R =   90.000 deg
};
P[2628]{
   GP1:
	UF : 0, UT : 6,		CONFIG : 'N U T, 0, 0, 0',
	X =  169.774  mm,	Y =   -449.820  mm,	Z =   -309.000  mm,
	W =  90.000 deg,	P =   0.000 deg,	R =   90.000 deg
};
P[2629]{
   GP1:
	UF : 0, UT : 6,		CONFIG : 'N U T, 0, 0, 0',
	X =  170.291  mm,	Y =   -450.307  mm,	Z =   -309.000  mm,
	W =  90.000 deg,	P =   0.000 deg,	R =   90.000 deg
};
P[2630]{
   GP1:
	UF : 0, UT : 6,		CONFIG : 'N U T, 0, 0, 0',
	X =  170.644  mm,	Y =   -449.167  mm,	Z =   -325.861  mm,
	W =  90.000 deg,	P =   0.000 deg,	R =   90.000 deg
};
P[2631]{
   GP1:
	UF : 0, UT : 6,		CONFIG : 'N U T, 0, 0, 0',
	X =  171.303  mm,	Y =   -449.791  mm,	Z =   -309.000  mm,
	W =  90.000 deg,	P =   0.000 deg,	R =   90.000 deg
};
P[2632]{
   GP1:
	UF : 0, UT : 6,		CONFIG : 'N U T, 0, 0, 0',
	X =  172.058  mm,	Y =   -448.936  mm,	Z =   -309.100  mm,
	W =  90.000 deg,	P =   0.000 deg,	R =   90.000 deg
};
P[2633]{
   GP1:
	UF : 0, UT : 6,		CONFIG : 'N U T, 0, 0, 0',
	X =  173.525  mm,	Y =   -447.991  mm,	Z =   -309.100  mm,
	W =  90.000 deg,	P =   0.000 deg,	R =   90.000 deg
};
P[2634]{
   GP1:
	UF : 0, UT : 6,		CONFIG : 'N U T, 0, 0, 0',
	X =  174.119  mm,	Y =   -447.617  mm,	Z =   -309.000  mm,
	W =  90.000 deg,	P =   0.000 deg,	R =   90.000 deg
};
P[2635]{
   GP1:
	UF : 0, UT : 6,		CONFIG : 'N U T, 0, 0, 0',
	X =  174.849  mm,	Y =   -447.825  mm,	Z =   -309.000  mm,
	W =  90.000 deg,	P =   0.000 deg,	R =   90.000 deg
};
P[2636]{
   GP1:
	UF : 0, UT : 6,		CONFIG : 'N U T, 0, 0, 0',
	X =  174.884  mm,	Y =   -446.670  mm,	Z =   -309.000  mm,
	W =  90.000 deg,	P =   0.000 deg,	R =   90.000 deg
};
P[2637]{
   GP1:
	UF : 0, UT : 6,		CONFIG : 'N U T, 0, 0, 0',
	X =  176.004  mm,	Y =   -446.723  mm,	Z =   -309.100  mm,
	W =  90.000 deg,	P =   0.000 deg,	R =   90.000 deg
};
P[2638]{
   GP1:
	UF : 0, UT : 6,		CONFIG : 'N U T, 0, 0, 0',
	X =  176.236  mm,	Y =   -446.098  mm,	Z =   -309.000  mm,
	W =  90.000 deg,	P =   0.000 deg,	R =   90.000 deg
};
P[2639]{
   GP1:
	UF : 0, UT : 6,		CONFIG : 'N U T, 0, 0, 0',
	X =  177.493  mm,	Y =   -445.997  mm,	Z =   -309.000  mm,
	W =  90.000 deg,	P =   0.000 deg,	R =   90.000 deg
};
P[2640]{
   GP1:
	UF : 0, UT : 6,		CONFIG : 'N U T, 0, 0, 0',
	X =  177.960  mm,	Y =   -445.068  mm,	Z =   -309.000  mm,
	W =  90.000 deg,	P =   0.000 deg,	R =   90.000 deg
};
P[2641]{
   GP1:
	UF : 0, UT : 6,		CONFIG : 'N U T, 0, 0, 0',
	X =  178.800  mm,	Y =   -445.033  mm,	Z =   -309.100  mm,
	W =  90.000 deg,	P =   0.000 deg,	R =   90.000 deg
};
P[2642]{
   GP1:
	UF : 0, UT : 6,		CONFIG : 'N U T, 0, 0, 0',
	X =  179.095  mm,	Y =   -444.399  mm,	Z =   -309.000  mm,
	W =  90.000 deg,	P =   0.000 deg,	R =   90.000 deg
};
P[2643]{
   GP1:
	UF : 0, UT : 6,		CONFIG : 'N U T, 0, 0, 0',
	X =  180.459  mm,	Y =   -444.217  mm,	Z =   -309.000  mm,
	W =  90.000 deg,	P =   0.000 deg,	R =   90.000 deg
};
P[2644]{
   GP1:
	UF : 0, UT : 6,		CONFIG : 'N U T, 0, 0, 0',
	X =  181.353  mm,	Y =   -443.920  mm,	Z =   -309.000  mm,
	W =  90.000 deg,	P =   0.000 deg,	R =   90.000 deg
};
P[2645]{
   GP1:
	UF : 0, UT : 6,		CONFIG : 'N U T, 0, 0, 0',
	X =  181.539  mm,	Y =   -442.927  mm,	Z =   -309.100  mm,
	W =  90.000 deg,	P =   0.000 deg,	R =   90.000 deg
};
P[2646]{
   GP1:
	UF : 0, UT : 6,		CONFIG : 'N U T, 0, 0, 0',
	X =  182.438  mm,	Y =   -443.166  mm,	Z =   -309.100  mm,
	W =  90.000 deg,	P =   0.000 deg,	R =   90.000 deg
};
P[2647]{
   GP1:
	UF : 0, UT : 6,		CONFIG : 'N U T, 0, 0, 0',
	X =  183.635  mm,	Y =   -442.374  mm,	Z =   -309.000  mm,
	W =  90.000 deg,	P =   0.000 deg,	R =   90.000 deg
};
P[2648]{
   GP1:
	UF : 0, UT : 6,		CONFIG : 'N U T, 0, 0, 0',
	X =  184.048  mm,	Y =   -441.662  mm,	Z =   -309.000  mm,
	W =  90.000 deg,	P =   0.000 deg,	R =   90.000 deg
};
P[2649]{
   GP1:
	UF : 0, UT : 6,		CONFIG : 'N U T, 0, 0, 0',
	X =  185.030  mm,	Y =   -441.468  mm,	Z =   -319.354  mm,
	W =  90.000 deg,	P =   0.000 deg,	R =   90.000 deg
};
P[2650]{
   GP1:
	UF : 0, UT : 6,		CONFIG : 'N U T, 0, 0, 0',
	X =  185.566  mm,	Y =   -440.824  mm,	Z =   -309.000  mm,
	W =  90.000 deg,	P =   0.000 deg,	R =   90.000 deg
};
P[2651]{
   GP1:
	UF : 0, UT : 6,		CONFIG : 'N U T, 0, 0, 0',
	X =  186.038  mm,	Y =   -441.372  mm,	Z =   -309.000  mm,
	W =  90.000 deg,	P =   0.000 deg,	R =   90.000 deg
};
P[2652]{
   GP1:
	UF : 0, UT : 6,		CONFIG : 'N U T, 0, 0, 0',
	X =  186.739  mm,	Y =   -440.764  mm,	Z =   -309.000  mm,
	W =  90.000 deg,	P =   0.000 deg,	R =   90.000 deg
};
P[2653]{
   GP1:
	UF : 0, UT : 6,		CONFIG : 'N U T, 0, 0, 0',
	X =  187.617  mm,	Y =   -439.990  mm,	Z =   -309.000  mm,
	W =  90.000 deg,	P =   0.000 deg,	R =   90.000 deg
};
P[2654]{
   GP1:
	UF : 0, UT : 6,		CONFIG : 'N U T, 0, 0, 0',
	X =  187.983  mm,	Y =   -439.402  mm,	Z =   -309.000  mm,
	W =  90.000 deg,	P =   0.000 deg,	R =   90.000 deg
};
P[2655]{
   GP1:
	UF : 0, UT : 6,		CONFIG : 'N U T, 0, 0, 0',
	X =  189.207  mm,	Y =   -439.108  mm,	Z =   -318.725  mm,
	W =  90.000 deg,	P =   0.000 deg,	R =   90.000 deg
};
P[2656]{
   GP1:
	UF : 0, UT : 6,		CONFIG : 'N U T, 0, 0, 0',
	X =  190.154  mm,	Y =   -438.352  mm,	Z =   -320.552  mm,
	W =  90.000 deg,	P =   0.000 deg,	R =   90.000 deg
};
P[2657]{
   GP1:
	UF : 0, UT : 6,		CONFIG : 'N U T, 0, 0, 0',
	X =  190.917  mm,	Y =   -437.476  mm,	Z =   -309.000  mm,
	W =  90.000 deg,	P =   0.000 deg,	R =   90.000 deg
};
P[2658]{
   GP1:
	UF : 0, UT : 6,		CONFIG : 'N U T, 0, 0, 0',
	X =  191.964  mm,	Y =   -437.572  mm,	Z =   -309.000  mm,
	W =  90.000 deg,	P =   0.000 deg,	R =   90.000 deg
};
P[2659]{
   GP1:
	UF : 0, UT : 6,		CONFIG : 'N U T, 0, 0, 0',
	X =  192.802  mm,	Y =   -436.893  mm,	Z =   -319.435  mm,
	W =  90.000 deg,	P =   0.000 deg,	R =   90.000 deg
};
P[2660]{
   GP1:
	UF : 0, UT : 6,		CONFIG : 'N U T, 0, 0, 0',
	X =  193.466  mm,	Y =   -436.104  mm,	Z =   -309.000  mm,
	W =  90.000 deg,	P =   0.000 deg,	R =   90.000 deg
};
P[2661]{
   GP1:
	UF : 0, UT : 6,		CONFIG : 'N U T, 0, 0, 0',
	X =  194.260  mm,	Y =   -436.251  mm,	Z =   -318.835  mm,
	W =  90.000 deg,	P =   0.000 deg,	R =   90.000 deg
};
P[2662]{
   GP1:
	UF : 0, UT : 6,		CONFIG : 'N U T, 0, 0, 0',
	X =  195.274  mm,	Y =   -435.488  mm,	Z =   -309.100  mm,
	W =  90.000 deg,	P =   0.000 deg,	R =   90.000 deg
};
P[2663]{
   GP1:
	UF : 0, UT : 6,		CONFIG : 'N U T, 0, 0, 0',
	X =  196.198  mm,	Y =   -434.698  mm,	Z =   -309.100  mm,
	W =  90.000 deg,	P =   0.000 deg,	R =   90.000 deg
};
P[2664]{
   GP1:
	UF : 0, UT : 6,		CONFIG : 'N U T, 0, 0, 0',
	X =  197.433  mm,	Y =   -434.097  mm,	Z =   -309.000  mm,
	W =  90.000 deg,	P =   0.000 deg,	R =   90.000 deg
};
P[2665]{
   GP1:
	UF : 0, UT : 6,		CONFIG : 'N U T, 0, 0, 0',
	X =  198.272  mm,	Y =   -434.197  mm,	Z =   -309.000  mm,
	W =  90.000 deg,	P =   0.000 deg,	R =   90.000 deg
};
P[2666]{
   GP1:
	UF : 0, UT : 6,		CONFIG : 'N U T, 0, 0, 0',
	X =  198.698  mm,	Y =   -433.197  mm,	Z =   -309.000  mm,
	W =  90.000 deg,	P =   0.000 deg,	R =   90.000 deg
};
P[2667]{
   GP1:
	UF : 0, UT : 6,		CONFIG : 'N U T, 0, 0, 0',
	X =  199.240  mm,	Y =   -433.329  mm,	Z =   -309.100  mm,
	W =  90.000 deg,	P =   0.000 deg,	R =   90.000 deg
};
P[2668]{
   GP1:
	UF : 0, UT : 6,		CONFIG : 'N U T, 0, 0, 0',
	X =  200.314  mm,	Y =   -433.071  mm,	Z =   -309.000  mm,
	W =  90.000 deg,	P =   0.000 deg,	R =   90.000 deg
};
P[2669]{
   GP1:
	UF : 0, UT : 6,		CONFIG : 'N U T, 0, 0, 0',
	X =  200.333  mm,	Y =   -432.385  mm,	Z =   -327.393  mm,
	W =  90.000 deg,	P =   0.000 deg,	R =   90.000 deg
};
P[2670]{
   GP1:
	UF : 0, UT : 6,		CONFIG : 'N U T, 0, 0, 0',
	X =  201.451  mm,	Y =   -432.237  mm,	Z =   -309.100  mm,
	W =  90.000 deg,	P =   0.000 deg,	R =   90.000 deg
};
P[2671]{
   GP1:
	UF : 0, UT : 6,		CONFIG : 'N U T, 0, 0, 0',
	X =  201.394  mm,	Y =   -431.387  mm,	Z =   -309.000  mm,
	W =  90.000 deg,	P =   0.000 deg,	R =   90.000 deg
};
P[2672]{
   GP1:
	UF : 0, UT : 6,		CONFIG : 'N U T, 0, 0, 0',
	X =  202.070  mm,	Y =   -431.372  mm,	Z =   -309.000  mm,
	W =  90.000 deg,	P =   0.000 deg,	R =   90.000 deg
};
P[2673]{
   GP1:
	UF : 0, UT : 6,		CONFIG : 'N U T, 0, 0, 0',
	X =  203.041  mm,	Y =   -430.798  mm,	Z =   -309.000  mm,
	W =  90.000 deg,	P =   0.000 deg,	R =   90.000 deg
};
P[2674]{
   GP1:
	UF : 0, UT : 6,		CONFIG : 'N U T, 0, 0, 0',
	X =  203.507  mm,	Y =   -430.984  mm,	Z =   -309.000  mm,
	W =  90.000 deg,	P =   0.000 deg,	R =   90.000 deg
};
P[2675]{
   GP1:
	UF : 0, UT : 6,		CONFIG : 'N U T, 0, 0, 0',
	X =  204.397  mm,	Y =   -430.559  mm,	Z =   -309.000  mm,
	W =  90.000 deg,	P =   0.000 deg,	R =   90.000 deg
};
P[2676]{
   GP1:
	UF : 0, UT : 6,		CONFIG : 'N U T, 0, 0, 0',
	X =  205.122  mm,	Y =   -429.883  mm,	Z =   -309.000  mm,
	W =  90.000 deg,	P =   0.000 deg,	R =   90.000 deg
};
P[2677]{
   GP1:
	UF : 0, UT : 6,		CONFIG : 'N U T, 0, 0, 0',
	X =  205.358  mm,	Y =   -429.138  mm,	Z =   -309.000  mm,
	W =  90.000 deg,	P =   0.000 deg,	R =   90.000 deg
};
P[2678]{
   GP1:
	UF : 0, UT : 6,		CONFIG : 'N U T, 0, 0, 0',
	X =  205.933  mm,	Y =   -429.606  mm,	Z =   -309.000  mm,
	W =  90.000 deg,	P =   0.000 deg,	R =   90.000 deg
};
P[2679]{
   GP1:
	UF : 0, UT : 6,		CONFIG : 'N U T, 0, 0, 0',
	X =  206.404  mm,	Y =   -428.744  mm,	Z =   -309.000  mm,
	W =  90.000 deg,	P =   0.000 deg,	R =   90.000 deg
};
P[2680]{
   GP1:
	UF : 0, UT : 6,		CONFIG : 'N U T, 0, 0, 0',
	X =  206.873  mm,	Y =   -429.098  mm,	Z =   -309.000  mm,
	W =  90.000 deg,	P =   0.000 deg,	R =   90.000 deg
};
P[2681]{
   GP1:
	UF : 0, UT : 6,		CONFIG : 'N U T, 0, 0, 0',
	X =  207.565  mm,	Y =   -428.300  mm,	Z =   -309.100  mm,
	W =  90.000 deg,	P =   0.000 deg,	R =   90.000 deg
};
P[2682]{
   GP1:
	UF : 0, UT : 6,		CONFIG : 'N U T, 0, 0, 0',
	X =  208.250  mm,	Y =   -427.928  mm,	Z =   -309.000  mm,
	W =  90.000 deg,	P =   0.000 deg,	R =   90.000 deg
};
P[2683]{
   GP1:
	UF : 0, UT : 6,		CONFIG : 'N U T, 0, 0, 0',
	X =  209.366  mm,	Y =   -427.616  mm,	Z =   -309.000  mm,
	W =  90.000 deg,	P =   0.000 deg,	R =   90.000 deg
};
P[2684]{
   GP1:
	UF : 0, UT : 6,		CONFIG : 'N U T, 0, 0, 0',
	X =  209.174  mm,	Y =   -426.878  mm,	Z =   -309.000  mm,
	W =  90.000 deg,	P =   0.000 deg,	R =   90.000 deg
};
P[2685]{
   GP1:
	UF : 0, UT : 6,		CONFIG : 'N U T, 0, 0, 0',
	X =  209.931  mm,	Y =   -426.841  mm,	Z =   -309.000  mm,
	W =  90.000 deg,	P =   0.000 deg,	R =   90.000 deg
};
P[2686]{
   GP1:
	UF : 0, UT : 6,		CONFIG : 'N U T, 0, 0, 0',
	X =  210.305  mm,	Y =   -427.095  mm,	Z =   -309.000  mm,
	W =  90.000 deg,	P =   0.000 deg,	R =   90.000 deg
};
P[2687]{
   GP1:
	UF : 0, UT : 6,		CONFIG : 'N U T, 0, 0, 0',
	X =  211.082  mm,	Y =   -426.149  mm,	Z =   -309.100  mm,
	W =  90.000 deg,	P =   0.000 deg,	R =   90.000 deg
};
P[2688]{
   GP1:
	UF : 0, UT : 6,		CONFIG : 'N U T, 0, 0, 0',
	X =  211.635  mm,	Y =   -426.360  mm,	Z =   -309.100  mm,
	W =  90.000 deg,	P =   0.000 deg,	R =   90.000 deg
};
P[2689]{
   GP1:
	UF : 0, UT : 6,		CONFIG : 'N U T, 0, 0, 0',
	X =  212.089  mm,	Y =   -425.910  mm,	Z =   -309.000  mm,
	W =  90.000 deg,	P =   0.000 deg,	R =   90.000 deg
};
P[2690]{
   GP1:
	UF : 0, UT : 6,		CONFIG : 'N U T, 0, 0, 0',
	X =  212.450  mm,	Y =   -425.742  mm,	Z =   -309.000  mm,
	W =  90.000 deg,	P =   0.000 deg,	R =   90.000 deg
};
P[2691]{
   GP1:
	UF : 0, UT : 6,		CONFIG : 'N U T, 0, 0, 0',
	X =  212.978  mm,	Y =   -425.408  mm,	Z =   -309.000  mm,
	W =  90.000 deg,	P =   0.000 deg,	R =   90.000 deg
};
P[2692]{
   GP1:
	UF : 0, UT : 6,		CONFIG : 'N U T, 0, 0, 0',
	X =  213.417  mm,	Y =   -425.007  mm,	Z =   -309.100  mm,
	W =  90.000 deg,	P =   0.000 deg,	R =   90.000 deg
};
P[2693]{
   GP1:
	UF : 0, UT : 6,		CONFIG : 'N U T, 0, 0, 0',
	X =  213.705  mm,	Y =   -425.283  mm,	Z =   -309.000  mm,
	W =  90.000 deg,	P =   0.000 deg,	R =   90.000 deg
};
P[2694]{
   GP1:
	UF : 0, UT : 6,		CONFIG : 'N U T, 0, 0, 0',
	X =  213.323  mm,	Y =   -424.601  mm,	Z =   -309.000  mm,
	W =  90.000 deg,	P =   0.000 deg,	R =   90.000 deg
};
P[2695]{
   GP1:
	UF : 0, UT : 6,		CONFIG : 'N U T, 0, 0, 0',
	X =  213.955  mm,	Y =   -424.986  mm,	Z =   -309.000  mm,
	W =  90.000 deg,	P =   0.000 deg,	R =   90.000 deg
};
P[2696]{
   GP1:
	UF : 0, UT : 6,		CONFIG : 'N U T, 0, 0, 0',
	X =  214.112  mm,	Y =   -424.395  mm,	Z =   -309.000  mm,
	W =  90.000 deg,	P =   0.000 deg,	R =   90.000 deg
};
P[2697]{
   GP1:
	UF : 0, UT : 6,		CONFIG : 'N U T, 0, 0, 0',
	X =  214.333  mm,	Y =   -424.668  mm,	Z =   -309.000  mm,
	W =  90.000 deg,	P =   0.000 deg,	R =   90.000 deg
};
P[2698]{
   GP1:
	UF : 0, UT : 6,		CONFIG : 'N U T, 0, 0, 0',
	X =  214.274  mm,	Y =   -424.385  mm,	Z =   -309.000  mm,
	W =  90.000 deg,	P =   0.000 deg,	R =   90.000 deg
};
P[2699]{
   GP1:
	UF : 0, UT : 6,		CONFIG : 'N U T, 0, 0, 0',
	X =  214.754  mm,	Y =   -424.144  mm,	Z =   -309.000  mm,
	W =  90.000 deg,	P =   0.000 deg,	R =   90.000 deg
};
P[2700]{
   GP1:
	UF : 0, UT : 6,		CONFIG : 'N U T, 0, 0, 0',
	X =  214.643  mm,	Y =   -423.927  mm,	Z =   -309.000  mm,
	W =  90.000 deg,	P =   0.000 deg,	R =   90.000 deg
};
P[2701]{
   GP1:
	UF : 0, UT : 6,		CONFIG : 'N U T, 0, 0, 0',
	X =  214.606  mm,	Y =   -423.834  mm,	Z =   -309.000  mm,
	W =  90.000 deg,	P =   0.000 deg,	R =   90.000 deg
};
P[2702]{
   GP1:
	UF : 0, UT : 6,		CONFIG : 'N U T, 0, 0, 0',
	X =  216.110  mm,	Y =   -423.593  mm,	Z =   -309.000  mm,
	W =  90.000 deg,	P =   0.000 deg,	R =   90.000 deg
};
P[2703]{
   GP1:
	UF : 0, UT : 6,		CONFIG : 'N U T, 0, 0, 0',
	X =  216.540  mm,	Y =   -422.955  mm,	Z =   -309.000  mm,
	W =  90.000 deg,	P =   0.000 deg,	R =   90.000 deg
};
P[2704]{
   GP1:
	UF : 0, UT : 6,		CONFIG : 'N U T, 0, 0, 0',
	X =  217.480  mm,	Y =   -422.611  mm,	Z =   -309.100  mm,
	W =  90.000 deg,	P =   0.000 deg,	R =   90.000 deg
};
P[2705]{
   GP1:
	UF : 0, UT : 6,		CONFIG : 'N U T, 0, 0, 0',
	X =  218.630  mm,	Y =   -421.784  mm,	Z =   -317.074  mm,
	W =  90.000 deg,	P =   0.000 deg,	R =   90.000 deg
};
P[2706]{
   GP1:
	UF : 0, UT : 6,		CONFIG : 'N U T, 0, 0, 0',
	X =  220.159  mm,	Y =   -420.621  mm,	Z =   -309.100  mm,
	W =  90.000 deg,	P =   0.000 deg,	R =   90.000 deg
};
P[2707]{
   GP1:
	UF : 0, UT : 6,		CONFIG : 'N U T, 0, 0, 0',
	X =  221.574  mm,	Y =   -420.215  mm,	Z =   -309.000  mm,
	W =  90.000 deg,	P =   0.000 deg,	R =   90.000 deg
};
P[2708]{
   GP1:
	UF : 0, UT : 6,		CONFIG : 'N U T, 0, 0, 0',
	X =  222.278  mm,	Y =   -420.044  mm,	Z =   -309.000  mm,
	W =  90.000 deg,	P =   0.000 deg,	R =   90.000 deg
};
P[2709]{
   GP1:
	UF : 0, UT : 6,		CONFIG : 'N U T, 0, 0, 0',
	X =  222.849  mm,	Y =   -419.498  mm,	Z =   -309.000  mm,
	W =  90.000 deg,	P =   0.000 deg,	R =   90.000 deg
};
P[2710]{
   GP1:
	UF : 0, UT : 6,		CONFIG : 'N U T, 0, 0, 0',
	X =  224.078  mm,	Y =   -418.659  mm,	Z =   -309.000  mm,
	W =  90.000 deg,	P =   0.000 deg,	R =   90.000 deg
};
P[2711]{
   GP1:
	UF : 0, UT : 6,		CONFIG : 'N U T, 0, 0, 0',
	X =  225.193  mm,	Y =   -418.411  mm,	Z =   -309.000  mm,
	W =  90.000 deg,	P =   0.000 deg,	R =   90.000 deg
};
P[2712]{
   GP1:
	UF : 0, UT : 6,		CONFIG : 'N U T, 0, 0, 0',
	X =  225.298  mm,	Y =   -417.611  mm,	Z =   -309.000  mm,
	W =  90.000 deg,	P =   0.000 deg,	R =   90.000 deg
};
P[2713]{
   GP1:
	UF : 0, UT : 6,		CONFIG : 'N U T, 0, 0, 0',
	X =  226.084  mm,	Y =   -417.632  mm,	Z =   -309.000  mm,
	W =  90.000 deg,	P =   0.000 deg,	R =   90.000 deg
};
P[2714]{
   GP1:
	UF : 0, UT : 6,		CONFIG : 'N U T, 0, 0, 0',
	X =  227.146  mm,	Y =   -417.394  mm,	Z =   -309.000  mm,
	W =  90.000 deg,	P =   0.000 deg,	R =   90.000 deg
};
P[2715]{
   GP1:
	UF : 0, UT : 6,		CONFIG : 'N U T, 0, 0, 0',
	X =  228.046  mm,	Y =   -416.780  mm,	Z =   -309.000  mm,
	W =  90.000 deg,	P =   0.000 deg,	R =   90.000 deg
};
P[2716]{
   GP1:
	UF : 0, UT : 6,		CONFIG : 'N U T, 0, 0, 0',
	X =  228.633  mm,	Y =   -415.952  mm,	Z =   -309.000  mm,
	W =  90.000 deg,	P =   0.000 deg,	R =   90.000 deg
};
P[2717]{
   GP1:
	UF : 0, UT : 6,		CONFIG : 'N U T, 0, 0, 0',
	X =  229.876  mm,	Y =   -415.043  mm,	Z =   -309.100  mm,
	W =  90.000 deg,	P =   0.000 deg,	R =   90.000 deg
};
P[2718]{
   GP1:
	UF : 0, UT : 6,		CONFIG : 'N U T, 0, 0, 0',
	X =  230.627  mm,	Y =   -415.027  mm,	Z =   -309.000  mm,
	W =  90.000 deg,	P =   0.000 deg,	R =   90.000 deg
};
P[2719]{
   GP1:
	UF : 0, UT : 6,		CONFIG : 'N U T, 0, 0, 0',
	X =  231.374  mm,	Y =   -414.121  mm,	Z =   -309.100  mm,
	W =  90.000 deg,	P =   0.000 deg,	R =   90.000 deg
};
P[2720]{
   GP1:
	UF : 0, UT : 6,		CONFIG : 'N U T, 0, 0, 0',
	X =  232.383  mm,	Y =   -414.270  mm,	Z =   -309.000  mm,
	W =  90.000 deg,	P =   0.000 deg,	R =   90.000 deg
};
P[2721]{
   GP1:
	UF : 0, UT : 6,		CONFIG : 'N U T, 0, 0, 0',
	X =  233.445  mm,	Y =   -413.613  mm,	Z =   -309.000  mm,
	W =  90.000 deg,	P =   0.000 deg,	R =   90.000 deg
};
P[2722]{
   GP1:
	UF : 0, UT : 6,		CONFIG : 'N U T, 0, 0, 0',
	X =  235.096  mm,	Y =   -412.528  mm,	Z =   -309.000  mm,
	W =  90.000 deg,	P =   0.000 deg,	R =   90.000 deg
};
P[2723]{
   GP1:
	UF : 0, UT : 6,		CONFIG : 'N U T, 0, 0, 0',
	X =  236.914  mm,	Y =   -411.516  mm,	Z =   -309.100  mm,
	W =  90.000 deg,	P =   0.000 deg,	R =   90.000 deg
};
P[2724]{
   GP1:
	UF : 0, UT : 6,		CONFIG : 'N U T, 0, 0, 0',
	X =  237.979  mm,	Y =   -410.964  mm,	Z =   -309.000  mm,
	W =  90.000 deg,	P =   0.000 deg,	R =   90.000 deg
};
P[2725]{
   GP1:
	UF : 0, UT : 6,		CONFIG : 'N U T, 0, 0, 0',
	X =  238.844  mm,	Y =   -410.359  mm,	Z =   -309.100  mm,
	W =  90.000 deg,	P =   0.000 deg,	R =   90.000 deg
};
P[2726]{
   GP1:
	UF : 0, UT : 6,		CONFIG : 'N U T, 0, 0, 0',
	X =  239.555  mm,	Y =   -410.124  mm,	Z =   -309.100  mm,
	W =  90.000 deg,	P =   0.000 deg,	R =   90.000 deg
};
P[2727]{
   GP1:
	UF : 0, UT : 6,		CONFIG : 'N U T, 0, 0, 0',
	X =  240.083  mm,	Y =   -409.530  mm,	Z =   -309.000  mm,
	W =  90.000 deg,	P =   0.000 deg,	R =   90.000 deg
};
P[2728]{
   GP1:
	UF : 0, UT : 6,		CONFIG : 'N U T, 0, 0, 0',
	X =  241.324  mm,	Y =   -409.162  mm,	Z =   -309.000  mm,
	W =  90.000 deg,	P =   0.000 deg,	R =   90.000 deg
};
P[2729]{
   GP1:
	UF : 0, UT : 6,		CONFIG : 'N U T, 0, 0, 0',
	X =  242.462  mm,	Y =   -408.240  mm,	Z =   -309.000  mm,
	W =  90.000 deg,	P =   0.000 deg,	R =   90.000 deg
};
P[2730]{
   GP1:
	UF : 0, UT : 6,		CONFIG : 'N U T, 0, 0, 0',
	X =  243.011  mm,	Y =   -407.372  mm,	Z =   -309.100  mm,
	W =  90.000 deg,	P =   0.000 deg,	R =   90.000 deg
};
P[2731]{
   GP1:
	UF : 0, UT : 6,		CONFIG : 'N U T, 0, 0, 0',
	X =  243.190  mm,	Y =   -407.597  mm,	Z =   -309.000  mm,
	W =  90.000 deg,	P =   0.000 deg,	R =   90.000 deg
};
P[2732]{
   GP1:
	UF : 0, UT : 6,		CONFIG : 'N U T, 0, 0, 0',
	X =  243.233  mm,	Y =   -407.673  mm,	Z =   -309.000  mm,
	W =  90.000 deg,	P =   0.000 deg,	R =   90.000 deg
};
P[2733]{
   GP1:
	UF : 0, UT : 6,		CONFIG : 'N U T, 0, 0, 0',
	X =  243.335  mm,	Y =   -407.849  mm,	Z =   -309.000  mm,
	W =  90.000 deg,	P =   0.000 deg,	R =   90.000 deg
};
P[2734]{
   GP1:
	UF : 0, UT : 6,		CONFIG : 'N U T, 0, 0, 0',
	X =  243.271  mm,	Y =   -407.605  mm,	Z =   -309.000  mm,
	W =  90.000 deg,	P =   0.000 deg,	R =   90.000 deg
};
P[2735]{
   GP1:
	UF : 0, UT : 6,		CONFIG : 'N U T, 0, 0, 0',
	X =  243.657  mm,	Y =   -408.102  mm,	Z =   -309.000  mm,
	W =  90.000 deg,	P =   0.000 deg,	R =   90.000 deg
};
P[2736]{
   GP1:
	UF : 0, UT : 6,		CONFIG : 'N U T, 0, 0, 0',
	X =  243.587  mm,	Y =   -407.060  mm,	Z =   -309.000  mm,
	W =  90.000 deg,	P =   0.000 deg,	R =   90.000 deg
};
P[2737]{
   GP1:
	UF : 0, UT : 6,		CONFIG : 'N U T, 0, 0, 0',
	X =  243.799  mm,	Y =   -407.425  mm,	Z =   -309.000  mm,
	W =  90.000 deg,	P =   0.000 deg,	R =   90.000 deg
};
P[2738]{
   GP1:
	UF : 0, UT : 6,		CONFIG : 'N U T, 0, 0, 0',
	X =  244.164  mm,	Y =   -406.832  mm,	Z =   -309.000  mm,
	W =  90.000 deg,	P =   0.000 deg,	R =   90.000 deg
};
P[2739]{
   GP1:
	UF : 0, UT : 6,		CONFIG : 'N U T, 0, 0, 0',
	X =  244.937  mm,	Y =   -406.805  mm,	Z =   -322.381  mm,
	W =  90.000 deg,	P =   0.000 deg,	R =   90.000 deg
};
P[2740]{
   GP1:
	UF : 0, UT : 6,		CONFIG : 'N U T, 0, 0, 0',
	X =  245.779  mm,	Y =   -406.210  mm,	Z =   -309.000  mm,
	W =  90.000 deg,	P =   0.000 deg,	R =   90.000 deg
};
P[2741]{
   GP1:
	UF : 0, UT : 6,		CONFIG : 'N U T, 0, 0, 0',
	X =  246.376  mm,	Y =   -406.364  mm,	Z =   -309.000  mm,
	W =  90.000 deg,	P =   0.000 deg,	R =   90.000 deg
};
P[2742]{
   GP1:
	UF : 0, UT : 6,		CONFIG : 'N U T, 0, 0, 0',
	X =  246.242  mm,	Y =   -405.713  mm,	Z =   -309.000  mm,
	W =  90.000 deg,	P =   0.000 deg,	R =   90.000 deg
};
P[2743]{
   GP1:
	UF : 0, UT : 6,		CONFIG : 'N U T, 0, 0, 0',
	X =  246.921  mm,	Y =   -405.545  mm,	Z =   -309.100  mm,
	W =  90.000 deg,	P =   0.000 deg,	R =   90.000 deg
};
P[2744]{
   GP1:
	UF : 0, UT : 6,		CONFIG : 'N U T, 0, 0, 0',
	X =  248.005  mm,	Y =   -405.304  mm,	Z =   -309.100  mm,
	W =  90.000 deg,	P =   0.000 deg,	R =   90.000 deg
};
P[2745]{
   GP1:
	UF : 0, UT : 6,		CONFIG : 'N U T, 0, 0, 0',
	X =  247.760  mm,	Y =   -404.604  mm,	Z =   -309.000  mm,
	W =  90.000 deg,	P =   0.000 deg,	R =   90.000 deg
};
P[2746]{
   GP1:
	UF : 0, UT : 6,		CONFIG : 'N U T, 0, 0, 0',
	X =  248.936  mm,	Y =   -404.226  mm,	Z =   -309.000  mm,
	W =  90.000 deg,	P =   0.000 deg,	R =   90.000 deg
};
P[2747]{
   GP1:
	UF : 0, UT : 6,		CONFIG : 'N U T, 0, 0, 0',
	X =  249.873  mm,	Y =   -403.737  mm,	Z =   -309.000  mm,
	W =  90.000 deg,	P =   0.000 deg,	R =   90.000 deg
};
P[2748]{
   GP1:
	UF : 0, UT : 6,		CONFIG : 'N U T, 0, 0, 0',
	X =  250.673  mm,	Y =   -403.569  mm,	Z =   -309.000  mm,
	W =  90.000 deg,	P =   0.000 deg,	R =   90.000 deg
};
P[2749]{
   GP1:
	UF : 0, UT : 6,		CONFIG : 'N U T, 0, 0, 0',
	X =  250.907  mm,	Y =   -402.890  mm,	Z =   -309.000  mm,
	W =  90.000 deg,	P =   0.000 deg,	R =   90.000 deg
};
P[2750]{
   GP1:
	UF : 0, UT : 6,		CONFIG : 'N U T, 0, 0, 0',
	X =  251.531  mm,	Y =   -403.430  mm,	Z =   -309.000  mm,
	W =  90.000 deg,	P =   0.000 deg,	R =   90.000 deg
};
P[2751]{
   GP1:
	UF : 0, UT : 6,		CONFIG : 'N U T, 0, 0, 0',
	X =  252.561  mm,	Y =   -402.906  mm,	Z =   -309.000  mm,
	W =  90.000 deg,	P =   0.000 deg,	R =   90.000 deg
};
P[2752]{
   GP1:
	UF : 0, UT : 6,		CONFIG : 'N U T, 0, 0, 0',
	X =  252.338  mm,	Y =   -402.210  mm,	Z =   -309.000  mm,
	W =  90.000 deg,	P =   0.000 deg,	R =   90.000 deg
};
P[2753]{
   GP1:
	UF : 0, UT : 6,		CONFIG : 'N U T, 0, 0, 0',
	X =  253.187  mm,	Y =   -402.151  mm,	Z =   -309.000  mm,
	W =  90.000 deg,	P =   0.000 deg,	R =   90.000 deg
};
P[2754]{
   GP1:
	UF : 0, UT : 6,		CONFIG : 'N U T, 0, 0, 0',
	X =  254.315  mm,	Y =   -401.443  mm,	Z =   -309.100  mm,
	W =  90.000 deg,	P =   0.000 deg,	R =   90.000 deg
};
P[2755]{
   GP1:
	UF : 0, UT : 6,		CONFIG : 'N U T, 0, 0, 0',
	X =  255.043  mm,	Y =   -401.046  mm,	Z =   -309.000  mm,
	W =  90.000 deg,	P =   0.000 deg,	R =   90.000 deg
};
P[2756]{
   GP1:
	UF : 0, UT : 6,		CONFIG : 'N U T, 0, 0, 0',
	X =  256.014  mm,	Y =   -400.866  mm,	Z =   -309.000  mm,
	W =  90.000 deg,	P =   0.000 deg,	R =   90.000 deg
};
P[2757]{
   GP1:
	UF : 0, UT : 6,		CONFIG : 'N U T, 0, 0, 0',
	X =  255.945  mm,	Y =   -400.285  mm,	Z =   -309.000  mm,
	W =  90.000 deg,	P =   0.000 deg,	R =   90.000 deg
};
P[2758]{
   GP1:
	UF : 0, UT : 6,		CONFIG : 'N U T, 0, 0, 0',
	X =  256.804  mm,	Y =   -400.513  mm,	Z =   -309.000  mm,
	W =  90.000 deg,	P =   0.000 deg,	R =   90.000 deg
};
P[2759]{
   GP1:
	UF : 0, UT : 6,		CONFIG : 'N U T, 0, 0, 0',
	X =  257.335  mm,	Y =   -399.600  mm,	Z =   -309.000  mm,
	W =  90.000 deg,	P =   0.000 deg,	R =   90.000 deg
};
P[2760]{
   GP1:
	UF : 0, UT : 6,		CONFIG : 'N U T, 0, 0, 0',
	X =  258.024  mm,	Y =   -398.698  mm,	Z =   -309.000  mm,
	W =  90.000 deg,	P =   0.000 deg,	R =   90.000 deg
};
P[2761]{
   GP1:
	UF : 0, UT : 6,		CONFIG : 'N U T, 0, 0, 0',
	X =  258.485  mm,	Y =   -399.209  mm,	Z =   -309.100  mm,
	W =  90.000 deg,	P =   0.000 deg,	R =   90.000 deg
};
P[2762]{
   GP1:
	UF : 0, UT : 6,		CONFIG : 'N U T, 0, 0, 0',
	X =  258.816  mm,	Y =   -398.272  mm,	Z =   -309.000  mm,
	W =  90.000 deg,	P =   0.000 deg,	R =   90.000 deg
};
P[2763]{
   GP1:
	UF : 0, UT : 6,		CONFIG : 'N U T, 0, 0, 0',
	X =  259.981  mm,	Y =   -397.719  mm,	Z =   -309.000  mm,
	W =  90.000 deg,	P =   0.000 deg,	R =   90.000 deg
};
P[2764]{
   GP1:
	UF : 0, UT : 6,		CONFIG : 'N U T, 0, 0, 0',
	X =  261.096  mm,	Y =   -397.314  mm,	Z =   -309.000  mm,
	W =  90.000 deg,	P =   0.000 deg,	R =   90.000 deg
};
P[2765]{
   GP1:
	UF : 0, UT : 6,		CONFIG : 'N U T, 0, 0, 0',
	X =  261.782  mm,	Y =   -396.995  mm,	Z =   -309.000  mm,
	W =  90.000 deg,	P =   0.000 deg,	R =   90.000 deg
};
P[2766]{
   GP1:
	UF : 0, UT : 6,		CONFIG : 'N U T, 0, 0, 0',
	X =  262.973  mm,	Y =   -396.678  mm,	Z =   -309.000  mm,
	W =  90.000 deg,	P =   0.000 deg,	R =   90.000 deg
};
P[2767]{
   GP1:
	UF : 0, UT : 6,		CONFIG : 'N U T, 0, 0, 0',
	X =  263.815  mm,	Y =   -396.402  mm,	Z =   -309.000  mm,
	W =  90.000 deg,	P =   0.000 deg,	R =   90.000 deg
};
P[2768]{
   GP1:
	UF : 0, UT : 6,		CONFIG : 'N U T, 0, 0, 0',
	X =  264.554  mm,	Y =   -395.999  mm,	Z =   -309.000  mm,
	W =  90.000 deg,	P =   0.000 deg,	R =   90.000 deg
};
P[2769]{
   GP1:
	UF : 0, UT : 6,		CONFIG : 'N U T, 0, 0, 0',
	X =  264.382  mm,	Y =   -395.248  mm,	Z =   -309.100  mm,
	W =  90.000 deg,	P =   0.000 deg,	R =   90.000 deg
};
P[2770]{
   GP1:
	UF : 0, UT : 6,		CONFIG : 'N U T, 0, 0, 0',
	X =  265.622  mm,	Y =   -395.097  mm,	Z =   -309.000  mm,
	W =  90.000 deg,	P =   0.000 deg,	R =   90.000 deg
};
P[2771]{
   GP1:
	UF : 0, UT : 6,		CONFIG : 'N U T, 0, 0, 0',
	X =  266.076  mm,	Y =   -394.168  mm,	Z =   -309.000  mm,
	W =  90.000 deg,	P =   0.000 deg,	R =   90.000 deg
};
P[2772]{
   GP1:
	UF : 0, UT : 6,		CONFIG : 'N U T, 0, 0, 0',
	X =  267.073  mm,	Y =   -393.984  mm,	Z =   -309.100  mm,
	W =  90.000 deg,	P =   0.000 deg,	R =   90.000 deg
};
P[2773]{
   GP1:
	UF : 0, UT : 6,		CONFIG : 'N U T, 0, 0, 0',
	X =  267.606  mm,	Y =   -393.411  mm,	Z =   -309.000  mm,
	W =  90.000 deg,	P =   0.000 deg,	R =   90.000 deg
};
P[2774]{
   GP1:
	UF : 0, UT : 6,		CONFIG : 'N U T, 0, 0, 0',
	X =  268.313  mm,	Y =   -393.630  mm,	Z =   -309.100  mm,
	W =  90.000 deg,	P =   0.000 deg,	R =   90.000 deg
};
P[2775]{
   GP1:
	UF : 0, UT : 6,		CONFIG : 'N U T, 0, 0, 0',
	X =  268.941  mm,	Y =   -393.149  mm,	Z =   -309.000  mm,
	W =  90.000 deg,	P =   0.000 deg,	R =   90.000 deg
};
P[2776]{
   GP1:
	UF : 0, UT : 6,		CONFIG : 'N U T, 0, 0, 0',
	X =  269.583  mm,	Y =   -392.172  mm,	Z =   -309.000  mm,
	W =  90.000 deg,	P =   0.000 deg,	R =   90.000 deg
};
P[2777]{
   GP1:
	UF : 0, UT : 6,		CONFIG : 'N U T, 0, 0, 0',
	X =  270.479  mm,	Y =   -392.196  mm,	Z =   -309.000  mm,
	W =  90.000 deg,	P =   0.000 deg,	R =   90.000 deg
};
P[2778]{
   GP1:
	UF : 0, UT : 6,		CONFIG : 'N U T, 0, 0, 0',
	X =  270.820  mm,	Y =   -391.528  mm,	Z =   -309.000  mm,
	W =  90.000 deg,	P =   0.000 deg,	R =   90.000 deg
};
P[2779]{
   GP1:
	UF : 0, UT : 6,		CONFIG : 'N U T, 0, 0, 0',
	X =  271.662  mm,	Y =   -391.446  mm,	Z =   -309.000  mm,
	W =  90.000 deg,	P =   0.000 deg,	R =   90.000 deg
};
P[2780]{
   GP1:
	UF : 0, UT : 6,		CONFIG : 'N U T, 0, 0, 0',
	X =  272.590  mm,	Y =   -390.908  mm,	Z =   -309.000  mm,
	W =  90.000 deg,	P =   0.000 deg,	R =   90.000 deg
};
P[2781]{
   GP1:
	UF : 0, UT : 6,		CONFIG : 'N U T, 0, 0, 0',
	X =  273.372  mm,	Y =   -389.976  mm,	Z =   -309.000  mm,
	W =  90.000 deg,	P =   0.000 deg,	R =   90.000 deg
};
P[2782]{
   GP1:
	UF : 0, UT : 6,		CONFIG : 'N U T, 0, 0, 0',
	X =  274.150  mm,	Y =   -390.166  mm,	Z =   -317.734  mm,
	W =  90.000 deg,	P =   0.000 deg,	R =   90.000 deg
};
P[2783]{
   GP1:
	UF : 0, UT : 6,		CONFIG : 'N U T, 0, 0, 0',
	X =  274.729  mm,	Y =   -389.354  mm,	Z =   -309.000  mm,
	W =  90.000 deg,	P =   0.000 deg,	R =   90.000 deg
};
P[2784]{
   GP1:
	UF : 0, UT : 6,		CONFIG : 'N U T, 0, 0, 0',
	X =  275.575  mm,	Y =   -389.339  mm,	Z =   -309.000  mm,
	W =  90.000 deg,	P =   0.000 deg,	R =   90.000 deg
};
P[2785]{
   GP1:
	UF : 0, UT : 6,		CONFIG : 'N U T, 0, 0, 0',
	X =  276.476  mm,	Y =   -388.634  mm,	Z =   -309.000  mm,
	W =  90.000 deg,	P =   0.000 deg,	R =   90.000 deg
};
P[2786]{
   GP1:
	UF : 0, UT : 6,		CONFIG : 'N U T, 0, 0, 0',
	X =  277.575  mm,	Y =   -388.060  mm,	Z =   -309.000  mm,
	W =  90.000 deg,	P =   0.000 deg,	R =   90.000 deg
};
P[2787]{
   GP1:
	UF : 0, UT : 6,		CONFIG : 'N U T, 0, 0, 0',
	X =  278.329  mm,	Y =   -387.349  mm,	Z =   -309.000  mm,
	W =  90.000 deg,	P =   0.000 deg,	R =   90.000 deg
};
P[2788]{
   GP1:
	UF : 0, UT : 6,		CONFIG : 'N U T, 0, 0, 0',
	X =  278.665  mm,	Y =   -387.848  mm,	Z =   -309.000  mm,
	W =  90.000 deg,	P =   0.000 deg,	R =   90.000 deg
};
P[2789]{
   GP1:
	UF : 0, UT : 6,		CONFIG : 'N U T, 0, 0, 0',
	X =  279.249  mm,	Y =   -386.730  mm,	Z =   -309.000  mm,
	W =  90.000 deg,	P =   0.000 deg,	R =   90.000 deg
};
P[2790]{
   GP1:
	UF : 0, UT : 6,		CONFIG : 'N U T, 0, 0, 0',
	X =  280.183  mm,	Y =   -386.598  mm,	Z =   -309.000  mm,
	W =  90.000 deg,	P =   0.000 deg,	R =   90.000 deg
};
P[2791]{
   GP1:
	UF : 0, UT : 6,		CONFIG : 'N U T, 0, 0, 0',
	X =  281.207  mm,	Y =   -385.404  mm,	Z =   -309.000  mm,
	W =  90.000 deg,	P =   0.000 deg,	R =   90.000 deg
};
P[2792]{
   GP1:
	UF : 0, UT : 6,		CONFIG : 'N U T, 0, 0, 0',
	X =  282.222  mm,	Y =   -385.247  mm,	Z =   -311.405  mm,
	W =  90.000 deg,	P =   0.000 deg,	R =   90.000 deg
};
P[2793]{
   GP1:
	UF : 0, UT : 6,		CONFIG : 'N U T, 0, 0, 0',
	X =  282.881  mm,	Y =   -384.876  mm,	Z =   -309.000  mm,
	W =  90.000 deg,	P =   0.000 deg,	R =   90.000 deg
};
P[2794]{
   GP1:
	UF : 0, UT : 6,		CONFIG : 'N U T, 0, 0, 0',
	X =  283.805  mm,	Y =   -384.344  mm,	Z =   -312.987  mm,
	W =  90.000 deg,	P =   0.000 deg,	R =   90.000 deg
};
P[2795]{
   GP1:
	UF : 0, UT : 6,		CONFIG : 'N U T, 0, 0, 0',
	X =  284.307  mm,	Y =   -383.773  mm,	Z =   -319.375  mm,
	W =  90.000 deg,	P =   0.000 deg,	R =   90.000 deg
};
P[2796]{
   GP1:
	UF : 0, UT : 6,		CONFIG : 'N U T, 0, 0, 0',
	X =  284.957  mm,	Y =   -383.591  mm,	Z =   -317.937  mm,
	W =  90.000 deg,	P =   0.000 deg,	R =   90.000 deg
};
P[2797]{
   GP1:
	UF : 0, UT : 6,		CONFIG : 'N U T, 0, 0, 0',
	X =  285.760  mm,	Y =   -383.532  mm,	Z =   -309.000  mm,
	W =  90.000 deg,	P =   0.000 deg,	R =   90.000 deg
};
P[2798]{
   GP1:
	UF : 0, UT : 6,		CONFIG : 'N U T, 0, 0, 0',
	X =  286.626  mm,	Y =   -382.631  mm,	Z =   -309.000  mm,
	W =  90.000 deg,	P =   0.000 deg,	R =   90.000 deg
};
P[2799]{
   GP1:
	UF : 0, UT : 6,		CONFIG : 'N U T, 0, 0, 0',
	X =  287.827  mm,	Y =   -382.240  mm,	Z =   -309.000  mm,
	W =  90.000 deg,	P =   0.000 deg,	R =   90.000 deg
};
P[2800]{
   GP1:
	UF : 0, UT : 6,		CONFIG : 'N U T, 0, 0, 0',
	X =  288.501  mm,	Y =   -381.826  mm,	Z =   -309.100  mm,
	W =  90.000 deg,	P =   0.000 deg,	R =   90.000 deg
};
P[2801]{
   GP1:
	UF : 0, UT : 6,		CONFIG : 'N U T, 0, 0, 0',
	X =  289.108  mm,	Y =   -381.645  mm,	Z =   -309.000  mm,
	W =  90.000 deg,	P =   0.000 deg,	R =   90.000 deg
};
P[2802]{
   GP1:
	UF : 0, UT : 6,		CONFIG : 'N U T, 0, 0, 0',
	X =  289.082  mm,	Y =   -380.937  mm,	Z =   -309.000  mm,
	W =  90.000 deg,	P =   0.000 deg,	R =   90.000 deg
};
P[2803]{
   GP1:
	UF : 0, UT : 6,		CONFIG : 'N U T, 0, 0, 0',
	X =  289.591  mm,	Y =   -381.071  mm,	Z =   -309.000  mm,
	W =  90.000 deg,	P =   0.000 deg,	R =   90.000 deg
};
P[2804]{
   GP1:
	UF : 0, UT : 6,		CONFIG : 'N U T, 0, 0, 0',
	X =  290.420  mm,	Y =   -381.011  mm,	Z =   -309.000  mm,
	W =  90.000 deg,	P =   0.000 deg,	R =   90.000 deg
};
P[2805]{
   GP1:
	UF : 0, UT : 6,		CONFIG : 'N U T, 0, 0, 0',
	X =  290.133  mm,	Y =   -380.377  mm,	Z =   -309.100  mm,
	W =  90.000 deg,	P =   0.000 deg,	R =   90.000 deg
};
P[2806]{
   GP1:
	UF : 0, UT : 6,		CONFIG : 'N U T, 0, 0, 0',
	X =  290.749  mm,	Y =   -379.777  mm,	Z =   -309.100  mm,
	W =  90.000 deg,	P =   0.000 deg,	R =   90.000 deg
};
P[2807]{
   GP1:
	UF : 0, UT : 6,		CONFIG : 'N U T, 0, 0, 0',
	X =  291.444  mm,	Y =   -379.901  mm,	Z =   -320.666  mm,
	W =  90.000 deg,	P =   0.000 deg,	R =   90.000 deg
};
P[2808]{
   GP1:
	UF : 0, UT : 6,		CONFIG : 'N U T, 0, 0, 0',
	X =  291.975  mm,	Y =   -380.034  mm,	Z =   -309.100  mm,
	W =  90.000 deg,	P =   0.000 deg,	R =   90.000 deg
};
P[2809]{
   GP1:
	UF : 0, UT : 6,		CONFIG : 'N U T, 0, 0, 0',
	X =  292.414  mm,	Y =   -379.141  mm,	Z =   -312.174  mm,
	W =  90.000 deg,	P =   0.000 deg,	R =   90.000 deg
};
P[2810]{
   GP1:
	UF : 0, UT : 6,		CONFIG : 'N U T, 0, 0, 0',
	X =  293.092  mm,	Y =   -379.153  mm,	Z =   -309.000  mm,
	W =  90.000 deg,	P =   0.000 deg,	R =   90.000 deg
};
P[2811]{
   GP1:
	UF : 0, UT : 6,		CONFIG : 'N U T, 0, 0, 0',
	X =  293.604  mm,	Y =   -378.481  mm,	Z =   -309.000  mm,
	W =  90.000 deg,	P =   0.000 deg,	R =   90.000 deg
};
P[2812]{
   GP1:
	UF : 0, UT : 6,		CONFIG : 'N U T, 0, 0, 0',
	X =  294.189  mm,	Y =   -378.377  mm,	Z =   -309.000  mm,
	W =  90.000 deg,	P =   0.000 deg,	R =   90.000 deg
};
P[2813]{
   GP1:
	UF : 0, UT : 6,		CONFIG : 'N U T, 0, 0, 0',
	X =  294.776  mm,	Y =   -377.892  mm,	Z =   -309.100  mm,
	W =  90.000 deg,	P =   0.000 deg,	R =   90.000 deg
};
P[2814]{
   GP1:
	UF : 0, UT : 6,		CONFIG : 'N U T, 0, 0, 0',
	X =  295.520  mm,	Y =   -377.457  mm,	Z =   -309.100  mm,
	W =  90.000 deg,	P =   0.000 deg,	R =   90.000 deg
};
P[2815]{
   GP1:
	UF : 0, UT : 6,		CONFIG : 'N U T, 0, 0, 0',
	X =  295.795  mm,	Y =   -377.557  mm,	Z =   -309.100  mm,
	W =  90.000 deg,	P =   0.000 deg,	R =   90.000 deg
};
P[2816]{
   GP1:
	UF : 0, UT : 6,		CONFIG : 'N U T, 0, 0, 0',
	X =  296.048  mm,	Y =   -377.630  mm,	Z =   -309.000  mm,
	W =  90.000 deg,	P =   0.000 deg,	R =   90.000 deg
};
P[2817]{
   GP1:
	UF : 0, UT : 6,		CONFIG : 'N U T, 0, 0, 0',
	X =  296.416  mm,	Y =   -377.287  mm,	Z =   -316.317  mm,
	W =  90.000 deg,	P =   0.000 deg,	R =   90.000 deg
};
P[2818]{
   GP1:
	UF : 0, UT : 6,		CONFIG : 'N U T, 0, 0, 0',
	X =  296.249  mm,	Y =   -376.916  mm,	Z =   -309.000  mm,
	W =  90.000 deg,	P =   0.000 deg,	R =   90.000 deg
};
P[2819]{
   GP1:
	UF : 0, UT : 6,		CONFIG : 'N U T, 0, 0, 0',
	X =  296.703  mm,	Y =   -377.454  mm,	Z =   -309.000  mm,
	W =  90.000 deg,	P =   0.000 deg,	R =   90.000 deg
};
P[2820]{
   GP1:
	UF : 0, UT : 6,		CONFIG : 'N U T, 0, 0, 0',
	X =  296.608  mm,	Y =   -377.159  mm,	Z =   -309.000  mm,
	W =  90.000 deg,	P =   0.000 deg,	R =   90.000 deg
};
P[2821]{
   GP1:
	UF : 0, UT : 6,		CONFIG : 'N U T, 0, 0, 0',
	X =  296.999  mm,	Y =   -376.170  mm,	Z =   -309.100  mm,
	W =  90.000 deg,	P =   0.000 deg,	R =   90.000 deg
};
P[2822]{
   GP1:
	UF : 0, UT : 6,		CONFIG : 'N U T, 0, 0, 0',
	X =  297.110  mm,	Y =   -376.304  mm,	Z =   -309.000  mm,
	W =  90.000 deg,	P =   0.000 deg,	R =   90.000 deg
};
P[2823]{
   GP1:
	UF : 0, UT : 6,		CONFIG : 'N U T, 0, 0, 0',
	X =  298.269  mm,	Y =   -376.145  mm,	Z =   -309.100  mm,
	W =  90.000 deg,	P =   0.000 deg,	R =   90.000 deg
};
P[2824]{
   GP1:
	UF : 0, UT : 6,		CONFIG : 'N U T, 0, 0, 0',
	X =  299.230  mm,	Y =   -375.463  mm,	Z =   -309.033  mm,
	W =  90.000 deg,	P =   0.000 deg,	R =   90.000 deg
};
P[2825]{
   GP1:
	UF : 0, UT : 6,		CONFIG : 'N U T, 0, 0, 0',
	X =  301.171  mm,	Y =   -374.165  mm,	Z =   -309.000  mm,
	W =  90.000 deg,	P =   0.000 deg,	R =   90.000 deg
};
P[2826]{
   GP1:
	UF : 0, UT : 6,		CONFIG : 'N U T, 0, 0, 0',
	X =  302.100  mm,	Y =   -373.639  mm,	Z =   -309.100  mm,
	W =  90.000 deg,	P =   0.000 deg,	R =   90.000 deg
};
P[2827]{
   GP1:
	UF : 0, UT : 6,		CONFIG : 'N U T, 0, 0, 0',
	X =  302.810  mm,	Y =   -373.504  mm,	Z =   -310.625  mm,
	W =  90.000 deg,	P =   0.000 deg,	R =   90.000 deg
};
P[2828]{
   GP1:
	UF : 0, UT : 6,		CONFIG : 'N U T, 0, 0, 0',
	X =  304.129  mm,	Y =   -372.680  mm,	Z =   -309.000  mm,
	W =  90.000 deg,	P =   0.000 deg,	R =   90.000 deg
};
P[2829]{
   GP1:
	UF : 0, UT : 6,		CONFIG : 'N U T, 0, 0, 0',
	X =  305.370  mm,	Y =   -372.193  mm,	Z =   -309.000  mm,
	W =  90.000 deg,	P =   0.000 deg,	R =   90.000 deg
};
P[2830]{
   GP1:
	UF : 0, UT : 6,		CONFIG : 'N U T, 0, 0, 0',
	X =  306.374  mm,	Y =   -371.546  mm,	Z =   -309.000  mm,
	W =  90.000 deg,	P =   0.000 deg,	R =   90.000 deg
};
P[2831]{
   GP1:
	UF : 0, UT : 6,		CONFIG : 'N U T, 0, 0, 0',
	X =  307.048  mm,	Y =   -370.361  mm,	Z =   -309.000  mm,
	W =  90.000 deg,	P =   0.000 deg,	R =   90.000 deg
};
P[2832]{
   GP1:
	UF : 0, UT : 6,		CONFIG : 'N U T, 0, 0, 0',
	X =  308.135  mm,	Y =   -370.591  mm,	Z =   -310.812  mm,
	W =  90.000 deg,	P =   0.000 deg,	R =   90.000 deg
};
P[2833]{
   GP1:
	UF : 0, UT : 6,		CONFIG : 'N U T, 0, 0, 0',
	X =  308.145  mm,	Y =   -369.817  mm,	Z =   -315.046  mm,
	W =  90.000 deg,	P =   0.000 deg,	R =   90.000 deg
};
P[2834]{
   GP1:
	UF : 0, UT : 6,		CONFIG : 'N U T, 0, 0, 0',
	X =  309.885  mm,	Y =   -369.277  mm,	Z =   -309.000  mm,
	W =  90.000 deg,	P =   0.000 deg,	R =   90.000 deg
};
P[2835]{
   GP1:
	UF : 0, UT : 6,		CONFIG : 'N U T, 0, 0, 0',
	X =  310.820  mm,	Y =   -369.046  mm,	Z =   -309.100  mm,
	W =  90.000 deg,	P =   0.000 deg,	R =   90.000 deg
};
P[2836]{
   GP1:
	UF : 0, UT : 6,		CONFIG : 'N U T, 0, 0, 0',
	X =  311.359  mm,	Y =   -368.548  mm,	Z =   -322.354  mm,
	W =  90.000 deg,	P =   0.000 deg,	R =   90.000 deg
};
P[2837]{
   GP1:
	UF : 0, UT : 6,		CONFIG : 'N U T, 0, 0, 0',
	X =  312.445  mm,	Y =   -368.216  mm,	Z =   -309.000  mm,
	W =  90.000 deg,	P =   0.000 deg,	R =   90.000 deg
};
P[2838]{
   GP1:
	UF : 0, UT : 6,		CONFIG : 'N U T, 0, 0, 0',
	X =  313.542  mm,	Y =   -367.591  mm,	Z =   -309.100  mm,
	W =  90.000 deg,	P =   0.000 deg,	R =   90.000 deg
};
P[2839]{
   GP1:
	UF : 0, UT : 6,		CONFIG : 'N U T, 0, 0, 0',
	X =  313.614  mm,	Y =   -366.707  mm,	Z =   -309.100  mm,
	W =  90.000 deg,	P =   0.000 deg,	R =   90.000 deg
};
P[2840]{
   GP1:
	UF : 0, UT : 6,		CONFIG : 'N U T, 0, 0, 0',
	X =  314.800  mm,	Y =   -366.456  mm,	Z =   -309.000  mm,
	W =  90.000 deg,	P =   0.000 deg,	R =   90.000 deg
};
P[2841]{
   GP1:
	UF : 0, UT : 6,		CONFIG : 'N U T, 0, 0, 0',
	X =  315.844  mm,	Y =   -366.229  mm,	Z =   -309.000  mm,
	W =  90.000 deg,	P =   0.000 deg,	R =   90.000 deg
};
P[2842]{
   GP1:
	UF : 0, UT : 6,		CONFIG : 'N U T, 0, 0, 0',
	X =  316.252  mm,	Y =   -365.111  mm,	Z =   -309.000  mm,
	W =  90.000 deg,	P =   0.000 deg,	R =   90.000 deg
};
P[2843]{
   GP1:
	UF : 0, UT : 6,		CONFIG : 'N U T, 0, 0, 0',
	X =  317.062  mm,	Y =   -365.126  mm,	Z =   -309.100  mm,
	W =  90.000 deg,	P =   0.000 deg,	R =   90.000 deg
};
P[2844]{
   GP1:
	UF : 0, UT : 6,		CONFIG : 'N U T, 0, 0, 0',
	X =  317.975  mm,	Y =   -364.535  mm,	Z =   -309.000  mm,
	W =  90.000 deg,	P =   0.000 deg,	R =   90.000 deg
};
P[2845]{
   GP1:
	UF : 0, UT : 6,		CONFIG : 'N U T, 0, 0, 0',
	X =  318.840  mm,	Y =   -364.360  mm,	Z =   -309.000  mm,
	W =  90.000 deg,	P =   0.000 deg,	R =   90.000 deg
};
P[2846]{
   GP1:
	UF : 0, UT : 6,		CONFIG : 'N U T, 0, 0, 0',
	X =  325.894  mm,	Y =   -377.265  mm,	Z =   -309.000  mm,
	W =  90.000 deg,	P =   0.000 deg,	R =   90.000 deg
};
P[2847]{
   GP1:
	UF : 0, UT : 6,		CONFIG : 'N U T, 0, 0, 0',
	X =  324.836  mm,	Y =   -377.958  mm,	Z =   -317.962  mm,
	W =  90.000 deg,	P =   0.000 deg,	R =   90.000 deg
};
P[2848]{
   GP1:
	UF : 0, UT : 6,		CONFIG : 'N U T, 0, 0, 0',
	X =  324.321  mm,	Y =   -378.467  mm,	Z =   -309.100  mm,
	W =  90.000 deg,	P =   0.000 deg,	R =   90.000 deg
};
P[2849]{
   GP1:
	UF : 0, UT : 6,		CONFIG : 'N U T, 0, 0, 0',
	X =  323.253  mm,	Y =   -378.987  mm,	Z =   -309.000  mm,
	W =  90.000 deg,	P =   0.000 deg,	R =   90.000 deg
};
P[2850]{
   GP1:
	UF : 0, UT : 6,		CONFIG : 'N U T, 0, 0, 0',
	X =  322.071  mm,	Y =   -379.085  mm,	Z =   -309.000  mm,
	W =  90.000 deg,	P =   0.000 deg,	R =   90.000 deg
};
P[2851]{
   GP1:
	UF : 0, UT : 6,		CONFIG : 'N U T, 0, 0, 0',
	X =  321.480  mm,	Y =   -380.095  mm,	Z =   -309.772  mm,
	W =  90.000 deg,	P =   0.000 deg,	R =   90.000 deg
};
P[2852]{
   GP1:
	UF : 0, UT : 6,		CONFIG : 'N U T, 0, 0, 0',
	X =  320.383  mm,	Y =   -381.124  mm,	Z =   -309.000  mm,
	W =  90.000 deg,	P =   0.000 deg,	R =   90.000 deg
};
P[2853]{
   GP1:
	UF : 0, UT : 6,		CONFIG : 'N U T, 0, 0, 0',
	X =  319.600  mm,	Y =   -380.916  mm,	Z =   -309.000  mm,
	W =  90.000 deg,	P =   0.000 deg,	R =   90.000 deg
};
P[2854]{
   GP1:
	UF : 0, UT : 6,		CONFIG : 'N U T, 0, 0, 0',
	X =  318.644  mm,	Y =   -382.115  mm,	Z =   -309.100  mm,
	W =  90.000 deg,	P =   0.000 deg,	R =   90.000 deg
};
P[2855]{
   GP1:
	UF : 0, UT : 6,		CONFIG : 'N U T, 0, 0, 0',
	X =  317.870  mm,	Y =   -382.082  mm,	Z =   -309.000  mm,
	W =  90.000 deg,	P =   0.000 deg,	R =   90.000 deg
};
P[2856]{
   GP1:
	UF : 0, UT : 6,		CONFIG : 'N U T, 0, 0, 0',
	X =  317.174  mm,	Y =   -382.492  mm,	Z =   -309.000  mm,
	W =  90.000 deg,	P =   0.000 deg,	R =   90.000 deg
};
P[2857]{
   GP1:
	UF : 0, UT : 6,		CONFIG : 'N U T, 0, 0, 0',
	X =  316.235  mm,	Y =   -382.390  mm,	Z =   -309.100  mm,
	W =  90.000 deg,	P =   0.000 deg,	R =   90.000 deg
};
P[2858]{
   GP1:
	UF : 0, UT : 6,		CONFIG : 'N U T, 0, 0, 0',
	X =  315.565  mm,	Y =   -383.527  mm,	Z =   -318.060  mm,
	W =  90.000 deg,	P =   0.000 deg,	R =   90.000 deg
};
P[2859]{
   GP1:
	UF : 0, UT : 6,		CONFIG : 'N U T, 0, 0, 0',
	X =  313.931  mm,	Y =   -383.875  mm,	Z =   -309.000  mm,
	W =  90.000 deg,	P =   0.000 deg,	R =   90.000 deg
};
P[2860]{
   GP1:
	UF : 0, UT : 6,		CONFIG : 'N U T, 0, 0, 0',
	X =  313.620  mm,	Y =   -384.669  mm,	Z =   -327.837  mm,
	W =  90.000 deg,	P =   0.000 deg,	R =   90.000 deg
};
P[2861]{
   GP1:
	UF : 0, UT : 6,		CONFIG : 'N U T, 0, 0, 0',
	X =  312.808  mm,	Y =   -385.023  mm,	Z =   -309.000  mm,
	W =  90.000 deg,	P =   0.000 deg,	R =   90.000 deg
};
P[2862]{
   GP1:
	UF : 0, UT : 6,		CONFIG : 'N U T, 0, 0, 0',
	X =  312.160  mm,	Y =   -385.818  mm,	Z =   -309.100  mm,
	W =  90.000 deg,	P =   0.000 deg,	R =   90.000 deg
};
P[2863]{
   GP1:
	UF : 0, UT : 6,		CONFIG : 'N U T, 0, 0, 0',
	X =  311.413  mm,	Y =   -385.845  mm,	Z =   -309.000  mm,
	W =  90.000 deg,	P =   0.000 deg,	R =   90.000 deg
};
P[2864]{
   GP1:
	UF : 0, UT : 6,		CONFIG : 'N U T, 0, 0, 0',
	X =  310.030  mm,	Y =   -386.320  mm,	Z =   -309.100  mm,
	W =  90.000 deg,	P =   0.000 deg,	R =   90.000 deg
};
P[2865]{
   GP1:
	UF : 0, UT : 6,		CONFIG : 'N U T, 0, 0, 0',
	X =  309.642  mm,	Y =   -387.097  mm,	Z =   -309.000  mm,
	W =  90.000 deg,	P =   0.000 deg,	R =   90.000 deg
};
P[2866]{
   GP1:
	UF : 0, UT : 6,		CONFIG : 'N U T, 0, 0, 0',
	X =  308.636  mm,	Y =   -387.502  mm,	Z =   -309.100  mm,
	W =  90.000 deg,	P =   0.000 deg,	R =   90.000 deg
};
P[2867]{
   GP1:
	UF : 0, UT : 6,		CONFIG : 'N U T, 0, 0, 0',
	X =  307.458  mm,	Y =   -387.781  mm,	Z =   -309.000  mm,
	W =  90.000 deg,	P =   0.000 deg,	R =   90.000 deg
};
P[2868]{
   GP1:
	UF : 0, UT : 6,		CONFIG : 'N U T, 0, 0, 0',
	X =  306.400  mm,	Y =   -388.333  mm,	Z =   -309.000  mm,
	W =  90.000 deg,	P =   0.000 deg,	R =   90.000 deg
};
P[2869]{
   GP1:
	UF : 0, UT : 6,		CONFIG : 'N U T, 0, 0, 0',
	X =  305.436  mm,	Y =   -388.702  mm,	Z =   -309.000  mm,
	W =  90.000 deg,	P =   0.000 deg,	R =   90.000 deg
};
P[2870]{
   GP1:
	UF : 0, UT : 6,		CONFIG : 'N U T, 0, 0, 0',
	X =  304.375  mm,	Y =   -389.507  mm,	Z =   -309.100  mm,
	W =  90.000 deg,	P =   0.000 deg,	R =   90.000 deg
};
P[2871]{
   GP1:
	UF : 0, UT : 6,		CONFIG : 'N U T, 0, 0, 0',
	X =  303.128  mm,	Y =   -390.602  mm,	Z =   -309.000  mm,
	W =  90.000 deg,	P =   0.000 deg,	R =   90.000 deg
};
P[2872]{
   GP1:
	UF : 0, UT : 6,		CONFIG : 'N U T, 0, 0, 0',
	X =  301.432  mm,	Y =   -391.383  mm,	Z =   -313.985  mm,
	W =  90.000 deg,	P =   0.000 deg,	R =   90.000 deg
};
P[2873]{
   GP1:
	UF : 0, UT : 6,		CONFIG : 'N U T, 0, 0, 0',
	X =  300.500  mm,	Y =   -392.359  mm,	Z =   -309.100  mm,
	W =  90.000 deg,	P =   0.000 deg,	R =   90.000 deg
};
P[2874]{
   GP1:
	UF : 0, UT : 6,		CONFIG : 'N U T, 0, 0, 0',
	X =  299.714  mm,	Y =   -392.713  mm,	Z =   -309.100  mm,
	W =  90.000 deg,	P =   0.000 deg,	R =   90.000 deg
};
P[2875]{
   GP1:
	UF : 0, UT : 6,		CONFIG : 'N U T, 0, 0, 0',
	X =  298.691  mm,	Y =   -393.462  mm,	Z =   -309.000  mm,
	W =  90.000 deg,	P =   0.000 deg,	R =   90.000 deg
};
P[2876]{
   GP1:
	UF : 0, UT : 6,		CONFIG : 'N U T, 0, 0, 0',
	X =  296.908  mm,	Y =   -394.083  mm,	Z =   -309.100  mm,
	W =  90.000 deg,	P =   0.000 deg,	R =   90.000 deg
};
P[2877]{
   GP1:
	UF : 0, UT : 6,		CONFIG : 'N U T, 0, 0, 0',
	X =  295.587  mm,	Y =   -394.918  mm,	Z =   -309.100  mm,
	W =  90.000 deg,	P =   0.000 deg,	R =   90.000 deg
};
P[2878]{
   GP1:
	UF : 0, UT : 6,		CONFIG : 'N U T, 0, 0, 0',
	X =  294.498  mm,	Y =   -395.408  mm,	Z =   -309.100  mm,
	W =  90.000 deg,	P =   0.000 deg,	R =   90.000 deg
};
P[2879]{
   GP1:
	UF : 0, UT : 6,		CONFIG : 'N U T, 0, 0, 0',
	X =  293.407  mm,	Y =   -395.803  mm,	Z =   -323.894  mm,
	W =  90.000 deg,	P =   0.000 deg,	R =   90.000 deg
};
P[2880]{
   GP1:
	UF : 0, UT : 6,		CONFIG : 'N U T, 0, 0, 0',
	X =  292.885  mm,	Y =   -396.377  mm,	Z =   -309.000  mm,
	W =  90.000 deg,	P =   0.000 deg,	R =   90.000 deg
};
P[2881]{
   GP1:
	UF : 0, UT : 6,		CONFIG : 'N U T, 0, 0, 0',
	X =  291.324  mm,	Y =   -397.024  mm,	Z =   -309.000  mm,
	W =  90.000 deg,	P =   0.000 deg,	R =   90.000 deg
};
P[2882]{
   GP1:
	UF : 0, UT : 6,		CONFIG : 'N U T, 0, 0, 0',
	X =  290.154  mm,	Y =   -397.789  mm,	Z =   -309.100  mm,
	W =  90.000 deg,	P =   0.000 deg,	R =   90.000 deg
};
P[2883]{
   GP1:
	UF : 0, UT : 6,		CONFIG : 'N U T, 0, 0, 0',
	X =  289.297  mm,	Y =   -398.801  mm,	Z =   -309.100  mm,
	W =  90.000 deg,	P =   0.000 deg,	R =   90.000 deg
};
P[2884]{
   GP1:
	UF : 0, UT : 6,		CONFIG : 'N U T, 0, 0, 0',
	X =  288.679  mm,	Y =   -399.182  mm,	Z =   -317.474  mm,
	W =  90.000 deg,	P =   0.000 deg,	R =   90.000 deg
};
P[2885]{
   GP1:
	UF : 0, UT : 6,		CONFIG : 'N U T, 0, 0, 0',
	X =  286.867  mm,	Y =   -399.946  mm,	Z =   -309.100  mm,
	W =  90.000 deg,	P =   0.000 deg,	R =   90.000 deg
};
P[2886]{
   GP1:
	UF : 0, UT : 6,		CONFIG : 'N U T, 0, 0, 0',
	X =  285.374  mm,	Y =   -400.235  mm,	Z =   -309.000  mm,
	W =  90.000 deg,	P =   0.000 deg,	R =   90.000 deg
};
P[2887]{
   GP1:
	UF : 0, UT : 6,		CONFIG : 'N U T, 0, 0, 0',
	X =  285.066  mm,	Y =   -400.908  mm,	Z =   -309.000  mm,
	W =  90.000 deg,	P =   0.000 deg,	R =   90.000 deg
};
P[2888]{
   GP1:
	UF : 0, UT : 6,		CONFIG : 'N U T, 0, 0, 0',
	X =  284.216  mm,	Y =   -401.413  mm,	Z =   -309.000  mm,
	W =  90.000 deg,	P =   0.000 deg,	R =   90.000 deg
};
P[2889]{
   GP1:
	UF : 0, UT : 6,		CONFIG : 'N U T, 0, 0, 0',
	X =  283.518  mm,	Y =   -401.746  mm,	Z =   -309.000  mm,
	W =  90.000 deg,	P =   0.000 deg,	R =   90.000 deg
};
P[2890]{
   GP1:
	UF : 0, UT : 6,		CONFIG : 'N U T, 0, 0, 0',
	X =  282.805  mm,	Y =   -402.332  mm,	Z =   -309.000  mm,
	W =  90.000 deg,	P =   0.000 deg,	R =   90.000 deg
};
P[2891]{
   GP1:
	UF : 0, UT : 6,		CONFIG : 'N U T, 0, 0, 0',
	X =  281.506  mm,	Y =   -402.970  mm,	Z =   -309.000  mm,
	W =  90.000 deg,	P =   0.000 deg,	R =   90.000 deg
};
P[2892]{
   GP1:
	UF : 0, UT : 6,		CONFIG : 'N U T, 0, 0, 0',
	X =  280.074  mm,	Y =   -403.637  mm,	Z =   -309.000  mm,
	W =  90.000 deg,	P =   0.000 deg,	R =   90.000 deg
};
P[2893]{
   GP1:
	UF : 0, UT : 6,		CONFIG : 'N U T, 0, 0, 0',
	X =  278.979  mm,	Y =   -404.285  mm,	Z =   -309.000  mm,
	W =  90.000 deg,	P =   0.000 deg,	R =   90.000 deg
};
P[2894]{
   GP1:
	UF : 0, UT : 6,		CONFIG : 'N U T, 0, 0, 0',
	X =  278.079  mm,	Y =   -405.507  mm,	Z =   -313.799  mm,
	W =  90.000 deg,	P =   0.000 deg,	R =   90.000 deg
};
P[2895]{
   GP1:
	UF : 0, UT : 6,		CONFIG : 'N U T, 0, 0, 0',
	X =  276.721  mm,	Y =   -405.760  mm,	Z =   -309.000  mm,
	W =  90.000 deg,	P =   0.000 deg,	R =   90.000 deg
};
P[2896]{
   GP1:
	UF : 0, UT : 6,		CONFIG : 'N U T, 0, 0, 0',
	X =  275.471  mm,	Y =   -406.392  mm,	Z =   -309.100  mm,
	W =  90.000 deg,	P =   0.000 deg,	R =   90.000 deg
};
P[2897]{
   GP1:
	UF : 0, UT : 6,		CONFIG : 'N U T, 0, 0, 0',
	X =  274.536  mm,	Y =   -407.064  mm,	Z =   -309.000  mm,
	W =  90.000 deg,	P =   0.000 deg,	R =   90.000 deg
};
P[2898]{
   GP1:
	UF : 0, UT : 6,		CONFIG : 'N U T, 0, 0, 0',
	X =  273.450  mm,	Y =   -407.800  mm,	Z =   -309.100  mm,
	W =  90.000 deg,	P =   0.000 deg,	R =   90.000 deg
};
P[2899]{
   GP1:
	UF : 0, UT : 6,		CONFIG : 'N U T, 0, 0, 0',
	X =  272.891  mm,	Y =   -408.501  mm,	Z =   -309.000  mm,
	W =  90.000 deg,	P =   0.000 deg,	R =   90.000 deg
};
P[2900]{
   GP1:
	UF : 0, UT : 6,		CONFIG : 'N U T, 0, 0, 0',
	X =  271.862  mm,	Y =   -408.771  mm,	Z =   -309.100  mm,
	W =  90.000 deg,	P =   0.000 deg,	R =   90.000 deg
};
P[2901]{
   GP1:
	UF : 0, UT : 6,		CONFIG : 'N U T, 0, 0, 0',
	X =  271.166  mm,	Y =   -408.459  mm,	Z =   -309.000  mm,
	W =  90.000 deg,	P =   0.000 deg,	R =   90.000 deg
};
P[2902]{
   GP1:
	UF : 0, UT : 6,		CONFIG : 'N U T, 0, 0, 0',
	X =  270.520  mm,	Y =   -409.120  mm,	Z =   -309.000  mm,
	W =  90.000 deg,	P =   0.000 deg,	R =   90.000 deg
};
P[2903]{
   GP1:
	UF : 0, UT : 6,		CONFIG : 'N U T, 0, 0, 0',
	X =  269.412  mm,	Y =   -410.009  mm,	Z =   -309.000  mm,
	W =  90.000 deg,	P =   0.000 deg,	R =   90.000 deg
};
P[2904]{
   GP1:
	UF : 0, UT : 6,		CONFIG : 'N U T, 0, 0, 0',
	X =  267.988  mm,	Y =   -410.337  mm,	Z =   -309.000  mm,
	W =  90.000 deg,	P =   0.000 deg,	R =   90.000 deg
};
P[2905]{
   GP1:
	UF : 0, UT : 6,		CONFIG : 'N U T, 0, 0, 0',
	X =  267.165  mm,	Y =   -411.287  mm,	Z =   -309.000  mm,
	W =  90.000 deg,	P =   0.000 deg,	R =   90.000 deg
};
P[2906]{
   GP1:
	UF : 0, UT : 6,		CONFIG : 'N U T, 0, 0, 0',
	X =  266.117  mm,	Y =   -412.034  mm,	Z =   -309.100  mm,
	W =  90.000 deg,	P =   0.000 deg,	R =   90.000 deg
};
P[2907]{
   GP1:
	UF : 0, UT : 6,		CONFIG : 'N U T, 0, 0, 0',
	X =  264.749  mm,	Y =   -412.315  mm,	Z =   -319.396  mm,
	W =  90.000 deg,	P =   0.000 deg,	R =   90.000 deg
};
P[2908]{
   GP1:
	UF : 0, UT : 6,		CONFIG : 'N U T, 0, 0, 0',
	X =  264.100  mm,	Y =   -412.833  mm,	Z =   -310.212  mm,
	W =  90.000 deg,	P =   0.000 deg,	R =   90.000 deg
};
P[2909]{
   GP1:
	UF : 0, UT : 6,		CONFIG : 'N U T, 0, 0, 0',
	X =  263.907  mm,	Y =   -413.609  mm,	Z =   -316.267  mm,
	W =  90.000 deg,	P =   0.000 deg,	R =   90.000 deg
};
P[2910]{
   GP1:
	UF : 0, UT : 6,		CONFIG : 'N U T, 0, 0, 0',
	X =  262.679  mm,	Y =   -413.954  mm,	Z =   -309.000  mm,
	W =  90.000 deg,	P =   0.000 deg,	R =   90.000 deg
};
P[2911]{
   GP1:
	UF : 0, UT : 6,		CONFIG : 'N U T, 0, 0, 0',
	X =  261.717  mm,	Y =   -414.469  mm,	Z =   -309.100  mm,
	W =  90.000 deg,	P =   0.000 deg,	R =   90.000 deg
};
P[2912]{
   GP1:
	UF : 0, UT : 6,		CONFIG : 'N U T, 0, 0, 0',
	X =  261.020  mm,	Y =   -415.345  mm,	Z =   -309.100  mm,
	W =  90.000 deg,	P =   0.000 deg,	R =   90.000 deg
};
P[2913]{
   GP1:
	UF : 0, UT : 6,		CONFIG : 'N U T, 0, 0, 0',
	X =  260.129  mm,	Y =   -415.714  mm,	Z =   -309.000  mm,
	W =  90.000 deg,	P =   0.000 deg,	R =   90.000 deg
};
P[2914]{
   GP1:
	UF : 0, UT : 6,		CONFIG : 'N U T, 0, 0, 0',
	X =  259.313  mm,	Y =   -416.353  mm,	Z =   -309.000  mm,
	W =  90.000 deg,	P =   0.000 deg,	R =   90.000 deg
};
P[2915]{
   GP1:
	UF : 0, UT : 6,		CONFIG : 'N U T, 0, 0, 0',
	X =  257.593  mm,	Y =   -416.911  mm,	Z =   -325.186  mm,
	W =  90.000 deg,	P =   0.000 deg,	R =   90.000 deg
};
P[2916]{
   GP1:
	UF : 0, UT : 6,		CONFIG : 'N U T, 0, 0, 0',
	X =  256.648  mm,	Y =   -417.366  mm,	Z =   -309.000  mm,
	W =  90.000 deg,	P =   0.000 deg,	R =   90.000 deg
};
P[2917]{
   GP1:
	UF : 0, UT : 6,		CONFIG : 'N U T, 0, 0, 0',
	X =  254.739  mm,	Y =   -418.454  mm,	Z =   -309.100  mm,
	W =  90.000 deg,	P =   0.000 deg,	R =   90.000 deg
};
P[2918]{
   GP1:
	UF : 0, UT : 6,		CONFIG : 'N U T, 0, 0, 0',
	X =  253.860  mm,	Y =   -418.851  mm,	Z =   -309.000  mm,
	W =  90.000 deg,	P =   0.000 deg,	R =   90.000 deg
};
P[2919]{
   GP1:
	UF : 0, UT : 6,		CONFIG : 'N U T, 0, 0, 0',
	X =  252.675  mm,	Y =   -419.154  mm,	Z =   -317.670  mm,
	W =  90.000 deg,	P =   0.000 deg,	R =   90.000 deg
};
P[2920]{
   GP1:
	UF : 0, UT : 6,		CONFIG : 'N U T, 0, 0, 0',
	X =  252.345  mm,	Y =   -420.221  mm,	Z =   -309.100  mm,
	W =  90.000 deg,	P =   0.000 deg,	R =   90.000 deg
};
P[2921]{
   GP1:
	UF : 0, UT : 6,		CONFIG : 'N U T, 0, 0, 0',
	X =  250.148  mm,	Y =   -420.747  mm,	Z =   -309.000  mm,
	W =  90.000 deg,	P =   0.000 deg,	R =   90.000 deg
};
P[2922]{
   GP1:
	UF : 0, UT : 6,		CONFIG : 'N U T, 0, 0, 0',
	X =  249.591  mm,	Y =   -421.288  mm,	Z =   -309.000  mm,
	W =  90.000 deg,	P =   0.000 deg,	R =   90.000 deg
};
P[2923]{
   GP1:
	UF : 0, UT : 6,		CONFIG : 'N U T, 0, 0, 0',
	X =  248.706  mm,	Y =   -422.011  mm,	Z =   -309.000  mm,
	W =  90.000 deg,	P =   0.000 deg,	R =   90.000 deg
};
P[2924]{
   GP1:
	UF : 0, UT : 6,		CONFIG : 'N U T, 0, 0, 0',
	X =  247.868  mm,	Y =   -422.486  mm,	Z =   -309.000  mm,
	W =  90.000 deg,	P =   0.000 deg,	R =   90.000 deg
};
P[2925]{
   GP1:
	UF : 0, UT : 6,		CONFIG : 'N U T, 0, 0, 0',
	X =  246.674  mm,	Y =   -422.742  mm,	Z =   -309.000  mm,
	W =  90.000 deg,	P =   0.000 deg,	R =   90.000 deg
};
P[2926]{
   GP1:
	UF : 0, UT : 6,		CONFIG : 'N U T, 0, 0, 0',
	X =  246.144  mm,	Y =   -423.732  mm,	Z =   -309.000  mm,
	W =  90.000 deg,	P =   0.000 deg,	R =   90.000 deg
};
P[2927]{
   GP1:
	UF : 0, UT : 6,		CONFIG : 'N U T, 0, 0, 0',
	X =  244.361  mm,	Y =   -424.627  mm,	Z =   -309.000  mm,
	W =  90.000 deg,	P =   0.000 deg,	R =   90.000 deg
};
P[2928]{
   GP1:
	UF : 0, UT : 6,		CONFIG : 'N U T, 0, 0, 0',
	X =  243.458  mm,	Y =   -425.162  mm,	Z =   -309.000  mm,
	W =  90.000 deg,	P =   0.000 deg,	R =   90.000 deg
};
P[2929]{
   GP1:
	UF : 0, UT : 6,		CONFIG : 'N U T, 0, 0, 0',
	X =  242.327  mm,	Y =   -425.170  mm,	Z =   -309.100  mm,
	W =  90.000 deg,	P =   0.000 deg,	R =   90.000 deg
};
P[2930]{
   GP1:
	UF : 0, UT : 6,		CONFIG : 'N U T, 0, 0, 0',
	X =  241.496  mm,	Y =   -426.540  mm,	Z =   -309.000  mm,
	W =  90.000 deg,	P =   0.000 deg,	R =   90.000 deg
};
P[2931]{
   GP1:
	UF : 0, UT : 6,		CONFIG : 'N U T, 0, 0, 0',
	X =  240.529  mm,	Y =   -426.332  mm,	Z =   -309.000  mm,
	W =  90.000 deg,	P =   0.000 deg,	R =   90.000 deg
};
P[2932]{
   GP1:
	UF : 0, UT : 6,		CONFIG : 'N U T, 0, 0, 0',
	X =  239.481  mm,	Y =   -426.804  mm,	Z =   -309.000  mm,
	W =  90.000 deg,	P =   0.000 deg,	R =   90.000 deg
};
P[2933]{
   GP1:
	UF : 0, UT : 6,		CONFIG : 'N U T, 0, 0, 0',
	X =  239.187  mm,	Y =   -427.602  mm,	Z =   -309.100  mm,
	W =  90.000 deg,	P =   0.000 deg,	R =   90.000 deg
};
P[2934]{
   GP1:
	UF : 0, UT : 6,		CONFIG : 'N U T, 0, 0, 0',
	X =  237.472  mm,	Y =   -428.548  mm,	Z =   -309.000  mm,
	W =  90.000 deg,	P =   0.000 deg,	R =   90.000 deg
};
P[2935]{
   GP1:
	UF : 0, UT : 6,		CONFIG : 'N U T, 0, 0, 0',
	X =  236.462  mm,	Y =   -428.855  mm,	Z =   -309.100  mm,
	W =  90.000 deg,	P =   0.000 deg,	R =   90.000 deg
};
P[2936]{
   GP1:
	UF : 0, UT : 6,		CONFIG : 'N U T, 0, 0, 0',
	X =  235.426  mm,	Y =   -429.297  mm,	Z =   -309.100  mm,
	W =  90.000 deg,	P =   0.000 deg,	R =   90.000 deg
};
P[2937]{
   GP1:
	UF : 0, UT : 6,		CONFIG : 'N U T, 0, 0, 0',
	X =  234.897  mm,	Y =   -430.194  mm,	Z =   -309.100  mm,
	W =  90.000 deg,	P =   0.000 deg,	R =   90.000 deg
};
P[2938]{
   GP1:
	UF : 0, UT : 6,		CONFIG : 'N U T, 0, 0, 0',
	X =  233.715  mm,	Y =   -430.584  mm,	Z =   -309.000  mm,
	W =  90.000 deg,	P =   0.000 deg,	R =   90.000 deg
};
P[2939]{
   GP1:
	UF : 0, UT : 6,		CONFIG : 'N U T, 0, 0, 0',
	X =  232.982  mm,	Y =   -430.761  mm,	Z =   -309.000  mm,
	W =  90.000 deg,	P =   0.000 deg,	R =   90.000 deg
};
P[2940]{
   GP1:
	UF : 0, UT : 6,		CONFIG : 'N U T, 0, 0, 0',
	X =  232.036  mm,	Y =   -431.769  mm,	Z =   -309.000  mm,
	W =  90.000 deg,	P =   0.000 deg,	R =   90.000 deg
};
P[2941]{
   GP1:
	UF : 0, UT : 6,		CONFIG : 'N U T, 0, 0, 0',
	X =  230.691  mm,	Y =   -432.442  mm,	Z =   -309.000  mm,
	W =  90.000 deg,	P =   0.000 deg,	R =   90.000 deg
};
P[2942]{
   GP1:
	UF : 0, UT : 6,		CONFIG : 'N U T, 0, 0, 0',
	X =  229.585  mm,	Y =   -433.117  mm,	Z =   -309.100  mm,
	W =  90.000 deg,	P =   0.000 deg,	R =   90.000 deg
};
P[2943]{
   GP1:
	UF : 0, UT : 6,		CONFIG : 'N U T, 0, 0, 0',
	X =  228.619  mm,	Y =   -433.645  mm,	Z =   -309.000  mm,
	W =  90.000 deg,	P =   0.000 deg,	R =   90.000 deg
};
P[2944]{
   GP1:
	UF : 0, UT : 6,		CONFIG : 'N U T, 0, 0, 0',
	X =  227.949  mm,	Y =   -433.550  mm,	Z =   -309.000  mm,
	W =  90.000 deg,	P =   0.000 deg,	R =   90.000 deg
};
P[2945]{
   GP1:
	UF : 0, UT : 6,		CONFIG : 'N U T, 0, 0, 0',
	X =  226.988  mm,	Y =   -434.470  mm,	Z =   -309.100  mm,
	W =  90.000 deg,	P =   0.000 deg,	R =   90.000 deg
};
P[2946]{
   GP1:
	UF : 0, UT : 6,		CONFIG : 'N U T, 0, 0, 0',
	X =  226.235  mm,	Y =   -434.730  mm,	Z =   -324.314  mm,
	W =  90.000 deg,	P =   0.000 deg,	R =   90.000 deg
};
P[2947]{
   GP1:
	UF : 0, UT : 6,		CONFIG : 'N U T, 0, 0, 0',
	X =  225.484  mm,	Y =   -435.336  mm,	Z =   -309.000  mm,
	W =  90.000 deg,	P =   0.000 deg,	R =   90.000 deg
};
P[2948]{
   GP1:
	UF : 0, UT : 6,		CONFIG : 'N U T, 0, 0, 0',
	X =  223.515  mm,	Y =   -436.420  mm,	Z =   -309.000  mm,
	W =  90.000 deg,	P =   0.000 deg,	R =   90.000 deg
};
P[2949]{
   GP1:
	UF : 0, UT : 6,		CONFIG : 'N U T, 0, 0, 0',
	X =  222.472  mm,	Y =   -437.456  mm,	Z =   -323.669  mm,
	W =  90.000 deg,	P =   0.000 deg,	R =   90.000 deg
};
P[2950]{
   GP1:
	UF : 0, UT : 6,		CONFIG : 'N U T, 0, 0, 0',
	X =  220.936  mm,	Y =   -438.140  mm,	Z =   -309.100  mm,
	W =  90.000 deg,	P =   0.000 deg,	R =   90.000 deg
};
P[2951]{
   GP1:
	UF : 0, UT : 6,		CONFIG : 'N U T, 0, 0, 0',
	X =  219.955  mm,	Y =   -438.270  mm,	Z =   -309.000  mm,
	W =  90.000 deg,	P =   0.000 deg,	R =   90.000 deg
};
P[2952]{
   GP1:
	UF : 0, UT : 6,		CONFIG : 'N U T, 0, 0, 0',
	X =  219.478  mm,	Y =   -438.994  mm,	Z =   -309.100  mm,
	W =  90.000 deg,	P =   0.000 deg,	R =   90.000 deg
};
P[2953]{
   GP1:
	UF : 0, UT : 6,		CONFIG : 'N U T, 0, 0, 0',
	X =  218.236  mm,	Y =   -439.245  mm,	Z =   -309.000  mm,
	W =  90.000 deg,	P =   0.000 deg,	R =   90.000 deg
};
P[2954]{
   GP1:
	UF : 0, UT : 6,		CONFIG : 'N U T, 0, 0, 0',
	X =  217.110  mm,	Y =   -439.851  mm,	Z =   -309.000  mm,
	W =  90.000 deg,	P =   0.000 deg,	R =   90.000 deg
};
P[2955]{
   GP1:
	UF : 0, UT : 6,		CONFIG : 'N U T, 0, 0, 0',
	X =  217.201  mm,	Y =   -440.627  mm,	Z =   -309.100  mm,
	W =  90.000 deg,	P =   0.000 deg,	R =   90.000 deg
};
P[2956]{
   GP1:
	UF : 0, UT : 6,		CONFIG : 'N U T, 0, 0, 0',
	X =  216.171  mm,	Y =   -441.123  mm,	Z =   -309.100  mm,
	W =  90.000 deg,	P =   0.000 deg,	R =   90.000 deg
};
P[2957]{
   GP1:
	UF : 0, UT : 6,		CONFIG : 'N U T, 0, 0, 0',
	X =  213.780  mm,	Y =   -441.547  mm,	Z =   -309.000  mm,
	W =  90.000 deg,	P =   0.000 deg,	R =   90.000 deg
};
P[2958]{
   GP1:
	UF : 0, UT : 6,		CONFIG : 'N U T, 0, 0, 0',
	X =  213.081  mm,	Y =   -442.515  mm,	Z =   -309.000  mm,
	W =  90.000 deg,	P =   0.000 deg,	R =   90.000 deg
};
P[2959]{
   GP1:
	UF : 0, UT : 6,		CONFIG : 'N U T, 0, 0, 0',
	X =  212.429  mm,	Y =   -442.884  mm,	Z =   -309.000  mm,
	W =  90.000 deg,	P =   0.000 deg,	R =   90.000 deg
};
P[2960]{
   GP1:
	UF : 0, UT : 6,		CONFIG : 'N U T, 0, 0, 0',
	X =  211.291  mm,	Y =   -443.441  mm,	Z =   -309.000  mm,
	W =  90.000 deg,	P =   0.000 deg,	R =   90.000 deg
};
P[2961]{
   GP1:
	UF : 0, UT : 6,		CONFIG : 'N U T, 0, 0, 0',
	X =  210.160  mm,	Y =   -444.021  mm,	Z =   -309.100  mm,
	W =  90.000 deg,	P =   0.000 deg,	R =   90.000 deg
};
P[2962]{
   GP1:
	UF : 0, UT : 6,		CONFIG : 'N U T, 0, 0, 0',
	X =  209.800  mm,	Y =   -444.682  mm,	Z =   -309.000  mm,
	W =  90.000 deg,	P =   0.000 deg,	R =   90.000 deg
};
P[2963]{
   GP1:
	UF : 0, UT : 6,		CONFIG : 'N U T, 0, 0, 0',
	X =  208.839  mm,	Y =   -445.010  mm,	Z =   -309.000  mm,
	W =  90.000 deg,	P =   0.000 deg,	R =   90.000 deg
};
P[2964]{
   GP1:
	UF : 0, UT : 6,		CONFIG : 'N U T, 0, 0, 0',
	X =  207.219  mm,	Y =   -445.959  mm,	Z =   -309.000  mm,
	W =  90.000 deg,	P =   0.000 deg,	R =   90.000 deg
};
P[2965]{
   GP1:
	UF : 0, UT : 6,		CONFIG : 'N U T, 0, 0, 0',
	X =  206.031  mm,	Y =   -446.480  mm,	Z =   -309.050  mm,
	W =  90.000 deg,	P =   0.000 deg,	R =   90.000 deg
};
P[2966]{
   GP1:
	UF : 0, UT : 6,		CONFIG : 'N U T, 0, 0, 0',
	X =  205.304  mm,	Y =   -447.051  mm,	Z =   -309.000  mm,
	W =  90.000 deg,	P =   0.000 deg,	R =   90.000 deg
};
P[2967]{
   GP1:
	UF : 0, UT : 6,		CONFIG : 'N U T, 0, 0, 0',
	X =  204.488  mm,	Y =   -447.244  mm,	Z =   -309.000  mm,
	W =  90.000 deg,	P =   0.000 deg,	R =   90.000 deg
};
P[2968]{
   GP1:
	UF : 0, UT : 6,		CONFIG : 'N U T, 0, 0, 0',
	X =  203.365  mm,	Y =   -447.996  mm,	Z =   -323.040  mm,
	W =  90.000 deg,	P =   0.000 deg,	R =   90.000 deg
};
P[2969]{
   GP1:
	UF : 0, UT : 6,		CONFIG : 'N U T, 0, 0, 0',
	X =  202.871  mm,	Y =   -448.578  mm,	Z =   -309.000  mm,
	W =  90.000 deg,	P =   0.000 deg,	R =   90.000 deg
};
P[2970]{
   GP1:
	UF : 0, UT : 6,		CONFIG : 'N U T, 0, 0, 0',
	X =  201.911  mm,	Y =   -449.188  mm,	Z =   -309.100  mm,
	W =  90.000 deg,	P =   0.000 deg,	R =   90.000 deg
};
P[2971]{
   GP1:
	UF : 0, UT : 6,		CONFIG : 'N U T, 0, 0, 0',
	X =  200.751  mm,	Y =   -449.609  mm,	Z =   -309.000  mm,
	W =  90.000 deg,	P =   0.000 deg,	R =   90.000 deg
};
P[2972]{
   GP1:
	UF : 0, UT : 6,		CONFIG : 'N U T, 0, 0, 0',
	X =  199.475  mm,	Y =   -450.416  mm,	Z =   -309.100  mm,
	W =  90.000 deg,	P =   0.000 deg,	R =   90.000 deg
};
P[2973]{
   GP1:
	UF : 0, UT : 6,		CONFIG : 'N U T, 0, 0, 0',
	X =  198.224  mm,	Y =   -450.766  mm,	Z =   -309.000  mm,
	W =  90.000 deg,	P =   0.000 deg,	R =   90.000 deg
};
P[2974]{
   GP1:
	UF : 0, UT : 6,		CONFIG : 'N U T, 0, 0, 0',
	X =  197.579  mm,	Y =   -451.305  mm,	Z =   -309.000  mm,
	W =  90.000 deg,	P =   0.000 deg,	R =   90.000 deg
};
P[2975]{
   GP1:
	UF : 0, UT : 6,		CONFIG : 'N U T, 0, 0, 0',
	X =  196.882  mm,	Y =   -451.594  mm,	Z =   -309.000  mm,
	W =  90.000 deg,	P =   0.000 deg,	R =   90.000 deg
};
P[2976]{
   GP1:
	UF : 0, UT : 6,		CONFIG : 'N U T, 0, 0, 0',
	X =  195.867  mm,	Y =   -452.664  mm,	Z =   -309.100  mm,
	W =  90.000 deg,	P =   0.000 deg,	R =   90.000 deg
};
P[2977]{
   GP1:
	UF : 0, UT : 6,		CONFIG : 'N U T, 0, 0, 0',
	X =  194.916  mm,	Y =   -453.443  mm,	Z =   -309.100  mm,
	W =  90.000 deg,	P =   0.000 deg,	R =   90.000 deg
};
P[2978]{
   GP1:
	UF : 0, UT : 6,		CONFIG : 'N U T, 0, 0, 0',
	X =  193.296  mm,	Y =   -453.854  mm,	Z =   -309.100  mm,
	W =  90.000 deg,	P =   0.000 deg,	R =   90.000 deg
};
P[2979]{
   GP1:
	UF : 0, UT : 6,		CONFIG : 'N U T, 0, 0, 0',
	X =  192.121  mm,	Y =   -454.696  mm,	Z =   -309.100  mm,
	W =  90.000 deg,	P =   0.000 deg,	R =   90.000 deg
};
P[2980]{
   GP1:
	UF : 0, UT : 6,		CONFIG : 'N U T, 0, 0, 0',
	X =  191.559  mm,	Y =   -455.124  mm,	Z =   -309.000  mm,
	W =  90.000 deg,	P =   0.000 deg,	R =   90.000 deg
};
P[2981]{
   GP1:
	UF : 0, UT : 6,		CONFIG : 'N U T, 0, 0, 0',
	X =  190.678  mm,	Y =   -455.635  mm,	Z =   -309.000  mm,
	W =  90.000 deg,	P =   0.000 deg,	R =   90.000 deg
};
P[2982]{
   GP1:
	UF : 0, UT : 6,		CONFIG : 'N U T, 0, 0, 0',
	X =  189.875  mm,	Y =   -455.895  mm,	Z =   -309.000  mm,
	W =  90.000 deg,	P =   0.000 deg,	R =   90.000 deg
};
P[2983]{
   GP1:
	UF : 0, UT : 6,		CONFIG : 'N U T, 0, 0, 0',
	X =  189.194  mm,	Y =   -456.314  mm,	Z =   -309.100  mm,
	W =  90.000 deg,	P =   0.000 deg,	R =   90.000 deg
};
P[2984]{
   GP1:
	UF : 0, UT : 6,		CONFIG : 'N U T, 0, 0, 0',
	X =  188.170  mm,	Y =   -457.155  mm,	Z =   -309.000  mm,
	W =  90.000 deg,	P =   0.000 deg,	R =   90.000 deg
};
P[2985]{
   GP1:
	UF : 0, UT : 6,		CONFIG : 'N U T, 0, 0, 0',
	X =  187.232  mm,	Y =   -457.519  mm,	Z =   -309.000  mm,
	W =  90.000 deg,	P =   0.000 deg,	R =   90.000 deg
};
P[2986]{
   GP1:
	UF : 0, UT : 6,		CONFIG : 'N U T, 0, 0, 0',
	X =  186.217  mm,	Y =   -457.773  mm,	Z =   -309.000  mm,
	W =  90.000 deg,	P =   0.000 deg,	R =   90.000 deg
};
P[2987]{
   GP1:
	UF : 0, UT : 6,		CONFIG : 'N U T, 0, 0, 0',
	X =  185.850  mm,	Y =   -458.604  mm,	Z =   -309.000  mm,
	W =  90.000 deg,	P =   0.000 deg,	R =   90.000 deg
};
P[2988]{
   GP1:
	UF : 0, UT : 6,		CONFIG : 'N U T, 0, 0, 0',
	X =  184.641  mm,	Y =   -458.790  mm,	Z =   -309.100  mm,
	W =  90.000 deg,	P =   0.000 deg,	R =   90.000 deg
};
P[2989]{
   GP1:
	UF : 0, UT : 6,		CONFIG : 'N U T, 0, 0, 0',
	X =  183.557  mm,	Y =   -459.285  mm,	Z =   -309.000  mm,
	W =  90.000 deg,	P =   0.000 deg,	R =   90.000 deg
};
P[2990]{
   GP1:
	UF : 0, UT : 6,		CONFIG : 'N U T, 0, 0, 0',
	X =  182.699  mm,	Y =   -460.268  mm,	Z =   -321.607  mm,
	W =  90.000 deg,	P =   0.000 deg,	R =   90.000 deg
};
P[2991]{
   GP1:
	UF : 0, UT : 6,		CONFIG : 'N U T, 0, 0, 0',
	X =  181.706  mm,	Y =   -460.498  mm,	Z =   -309.000  mm,
	W =  90.000 deg,	P =   0.000 deg,	R =   90.000 deg
};
P[2992]{
   GP1:
	UF : 0, UT : 6,		CONFIG : 'N U T, 0, 0, 0',
	X =  180.267  mm,	Y =   -461.421  mm,	Z =   -309.000  mm,
	W =  90.000 deg,	P =   0.000 deg,	R =   90.000 deg
};
P[2993]{
   GP1:
	UF : 0, UT : 6,		CONFIG : 'N U T, 0, 0, 0',
	X =  179.424  mm,	Y =   -461.867  mm,	Z =   -309.100  mm,
	W =  90.000 deg,	P =   0.000 deg,	R =   90.000 deg
};
P[2994]{
   GP1:
	UF : 0, UT : 6,		CONFIG : 'N U T, 0, 0, 0',
	X =  178.726  mm,	Y =   -462.436  mm,	Z =   -309.100  mm,
	W =  90.000 deg,	P =   0.000 deg,	R =   90.000 deg
};
P[2995]{
   GP1:
	UF : 0, UT : 6,		CONFIG : 'N U T, 0, 0, 0',
	X =  177.739  mm,	Y =   -463.045  mm,	Z =   -309.100  mm,
	W =  90.000 deg,	P =   0.000 deg,	R =   90.000 deg
};
P[2996]{
   GP1:
	UF : 0, UT : 6,		CONFIG : 'N U T, 0, 0, 0',
	X =  176.133  mm,	Y =   -464.065  mm,	Z =   -309.100  mm,
	W =  90.000 deg,	P =   0.000 deg,	R =   90.000 deg
};
P[2997]{
   GP1:
	UF : 0, UT : 6,		CONFIG : 'N U T, 0, 0, 0',
	X =  175.309  mm,	Y =   -464.402  mm,	Z =   -309.100  mm,
	W =  90.000 deg,	P =   0.000 deg,	R =   90.000 deg
};
P[2998]{
   GP1:
	UF : 0, UT : 6,		CONFIG : 'N U T, 0, 0, 0',
	X =  174.296  mm,	Y =   -464.821  mm,	Z =   -309.000  mm,
	W =  90.000 deg,	P =   0.000 deg,	R =   90.000 deg
};
P[2999]{
   GP1:
	UF : 0, UT : 6,		CONFIG : 'N U T, 0, 0, 0',
	X =  173.412  mm,	Y =   -465.439  mm,	Z =   -309.100  mm,
	W =  90.000 deg,	P =   0.000 deg,	R =   90.000 deg
};
P[3000]{
   GP1:
	UF : 0, UT : 6,		CONFIG : 'N U T, 0, 0, 0',
	X =  172.624  mm,	Y =   -466.409  mm,	Z =   -311.033  mm,
	W =  90.000 deg,	P =   0.000 deg,	R =   90.000 deg
};
P[3001]{
   GP1:
	UF : 0, UT : 6,		CONFIG : 'N U T, 0, 0, 0',
	X =  171.546  mm,	Y =   -466.198  mm,	Z =   -309.100  mm,
	W =  90.000 deg,	P =   0.000 deg,	R =   90.000 deg
};
P[3002]{
   GP1:
	UF : 0, UT : 6,		CONFIG : 'N U T, 0, 0, 0',
	X =  170.479  mm,	Y =   -467.129  mm,	Z =   -309.000  mm,
	W =  90.000 deg,	P =   0.000 deg,	R =   90.000 deg
};
P[3003]{
   GP1:
	UF : 0, UT : 6,		CONFIG : 'N U T, 0, 0, 0',
	X =  169.803  mm,	Y =   -467.461  mm,	Z =   -309.000  mm,
	W =  90.000 deg,	P =   0.000 deg,	R =   90.000 deg
};
P[3004]{
   GP1:
	UF : 0, UT : 6,		CONFIG : 'N U T, 0, 0, 0',
	X =  168.884  mm,	Y =   -467.840  mm,	Z =   -309.000  mm,
	W =  90.000 deg,	P =   0.000 deg,	R =   90.000 deg
};
P[3005]{
   GP1:
	UF : 0, UT : 6,		CONFIG : 'N U T, 0, 0, 0',
	X =  168.245  mm,	Y =   -468.477  mm,	Z =   -309.000  mm,
	W =  90.000 deg,	P =   0.000 deg,	R =   90.000 deg
};
P[3006]{
   GP1:
	UF : 0, UT : 6,		CONFIG : 'N U T, 0, 0, 0',
	X =  167.152  mm,	Y =   -468.871  mm,	Z =   -309.000  mm,
	W =  90.000 deg,	P =   0.000 deg,	R =   90.000 deg
};
P[3007]{
   GP1:
	UF : 0, UT : 6,		CONFIG : 'N U T, 0, 0, 0',
